// Check ParCmd.ProcessingMode defined ? 
IF (( ProcessingMode < ProcessingModeEnum.BUFFERED         ) AND
    ( ProcessingMode > ProcessingModeEnum.TRIGGER_MULTIPLE ))
THEN
  // Parameter not valid
  CheckParameterValid := FALSE;
  // Set error
  SetError( ErrorID := RobotLibraryErrorIdEnum.ERR_PROCESSINGMODE_NOT_DEFINED, Overwrite := TRUE );
  // Create log entry
  CreateLogMessagePara1 ( Timestamp   := AxesGroup.State.SystemTime,
                          MessageType := MessageType.CMD,
                          Severity    := Severity.ERROR,
                          MessageCode := ErrorID,
                          MessageText := 'Invalid Parameter ParCmd.ProcessingMode = {1}',
                          Para1       := PROCESSING_MODE_TO_STRING(ProcessingMode));
  RETURN;                          
END_IF


// Check ProcessingMode valid ? 
IF (( ProcessingMode <> ProcessingModeEnum.BUFFERED           ) AND
    ( ProcessingMode <> ProcessingModeEnum.ABORTING           ) AND  
    ( ProcessingMode <> ProcessingModeEnum.PARALLEL           ) AND
    ( ProcessingMode <> ProcessingModeEnum.CONTINUOUS         ) AND
    ( ProcessingMode <> ProcessingModeEnum.DEACTIVATE         ) AND
    ( ProcessingMode <> ProcessingModeEnum.TRIGGER_ONCE       ) AND
    ( ProcessingMode <> ProcessingModeEnum.TRIGGER_CONTINUOUS ) AND
    ( ProcessingMode <> ProcessingModeEnum.TRIGGER_MULTIPLE   )) 
THEN
  // Parameter not valid
  CheckParameterValid := FALSE;
  // Set error
  SetError( ErrorID := RobotLibraryErrorIdEnum.ERR_PROCESSINGMODE_NOT_ALLOWED, Overwrite := TRUE );
  // Create log entry
  CreateLogMessagePara1 ( Timestamp   := AxesGroup.State.SystemTime,
                          MessageType := MessageType.CMD,
                          Severity    := Severity.ERROR,
                          MessageCode := ErrorID,
                          MessageText := 'Invalid Parameter ProcessingMode = {1}',
                          Para1       := PROCESSING_MODE_TO_STRING(ProcessingMode));
  RETURN;                          
END_IF

// Check SequenceFlag valid ? 
IF (( SequenceFlag <> SequenceFlagEnum.NO_SEQUENCE        ) AND    
    ( SequenceFlag <> SequenceFlagEnum.PRIMARY_SEQUENCE   ) AND
    ( SequenceFlag <> SequenceFlagEnum.SECONDARY_SEQUENCE ))
THEN
  // Parameter not valid
  CheckParameterValid := FALSE;
  // Set error
  SetError( ErrorID := RobotLibraryErrorIdEnum.ERR_SEQFLAG_NOT_ALLOWED, Overwrite := TRUE );
  // Create log entry
  CreateLogMessagePara1 ( Timestamp   := AxesGroup.State.SystemTime,
                          MessageType := MessageType.CMD,
                          Severity    := Severity.ERROR,
                          MessageCode := ErrorID,
                          MessageText := 'Invalid Parameter SequenceFlag = {1}',
                          Para1       := SEQUENCE_FLAG_TO_STRING(SequenceFlag));
  RETURN;                          
END_IF


// Check ParCmd.JobID valid ? 
IF (( ParCmd.JobID <     0 ) OR  
    ( ParCmd.JobID > 65535 ))
THEN
  // Parameter not valid
  CheckParameterValid := FALSE;
  // Set error
  SetError( ErrorID := RobotLibraryErrorIdEnum.ERR_LISTENERID_MUST_BE_POSITIVE, Overwrite := TRUE );
  // Create log entry
  CreateLogMessagePara1 ( Timestamp   := AxesGroup.State.SystemTime,
                          MessageType := MessageType.CMD,
                          Severity    := Severity.ERROR,
                          MessageCode := ErrorID,
                          MessageText := 'Invalid Parameter ParCmd.JobID = {1}',
                          Para1       := UINT_TO_STRING(ParCmd.JobID));
  RETURN;                          
END_IF


// Check ParCmd.ListenerID valid ? 
IF (( ParCmd.ListenerID <   0 ) OR  
    ( ParCmd.ListenerID > 127 ))
THEN
  // Parameter not valid
  CheckParameterValid := FALSE;
  // Set error
  SetError( ErrorID := RobotLibraryErrorIdEnum.ERR_LISTENERID_MUST_BE_POSITIVE, Overwrite := TRUE );
  // Create log entry
  CreateLogMessagePara1 ( Timestamp   := AxesGroup.State.SystemTime,
                          MessageType := MessageType.CMD,
                          Severity    := Severity.ERROR,
                          MessageCode := ErrorID,
                          MessageText := 'Invalid Parameter ParCmd.ListenerID = {1}',
                          Para1       := SINT_TO_STRING(ParCmd.ListenerID));
  RETURN;                          
END_IF



FOR _idx := 0 TO RobotLibraryParameter.SUB_PROGRAM_DATA_MAX
DO
  // Check ParCmd.Data valid ? 
  IF (( ParCmd.Data[_idx] <   0 ) OR  
      ( ParCmd.Data[_idx] > 255 ))
  THEN
    // Parameter not valid
    CheckParameterValid := FALSE;
    // Set error
    SetError( ErrorID := RobotLibraryErrorIdEnum.ERR_LISTENERID_MUST_BE_POSITIVE, Overwrite := TRUE );
    // Create log entry
    CreateLogMessagePara2 ( Timestamp   := AxesGroup.State.SystemTime,
                            MessageType := MessageType.CMD,
                            Severity    := Severity.ERROR,
                            MessageCode := ErrorID,
                            MessageText := 'Invalid Parameter ParCmd.Data[{2}] = {1}',
                            Para1       := BYTE_TO_STRING(ParCmd.Data[_idx]),
                            Para2       := DINT_TO_STRING(_idx));
    EXIT;                            
    RETURN;                          
  END_IF
END_FOR
                
END_METHOD

METHOD INTERNAL CreateCommandPayload : RobotLibraryCommandDataFB
VAR_IN_OUT
  /// Robot assignment of function
  AxesGroup : AxesGroup; 
END_VAR
VAR
  /// internal index for loops
 _idx          : DINT;
  /// Parameter count
 _parameterCnt : DINT;
END_VAR// Table 6-687: Sent CMD payload (PLC to RC) of "CallSubprogram"
// --------------------------
// Header
// --------------------------
// Byte 00 : UINT  - Type HB     
// Byte 01 :       - Type LB    
// Byte 02 : USINT - Reserve | ExecutionMode
// Byte 03 : USINT - ParSeq  | Priority
// --------------------------
// Datablock
// --------------------------
// Byte 00 : UINT  Type;
// Byte 01 :       Type;
// Byte 02 : USINT Reserved ExecutionMode;
// Byte 03 : USINT ParSeq Priority;
// Byte 04 : SINT  EmitterID[0];
// Byte 05 : SINT  EmitterID[1];
// Byte 06 : SINT  EmitterID[2];
// Byte 07 : SINT  EmitterID[3];
// Byte 08 : SINT  ListenerID;
// Byte 09 : BYTE  Reserved;
// Byte 10 : UINT  JobID;
// Byte 11 :       JobID;
// Byte 12 : BYTE  Data[0];
// Byte 13 : BYTE  Data[1];
// Byte 14 : BYTE  Data[2];
// Byte 15 : BYTE  Data[3];
// Byte 16 : BYTE  Data[4];
// Byte 17 : BYTE  Data[5];
// Byte 18 : BYTE  Data[6];
// Byte 19 : BYTE  Data[7];
// Byte 20 : BYTE  Data[8];
// Byte 21 : BYTE  Data[9];
// Byte 22 : BYTE  Data[10];
// Byte 23 : BYTE  Data[11];
// Byte 24 : BYTE  Data[12];
// Byte 25 : BYTE  Data[13];
// Byte 26 : BYTE  Data[14];
// Byte 27 : BYTE  Data[15];
// Byte 28 : BYTE  Data[16];
// Byte 29 : BYTE  Data[17];
// Byte 30 : BYTE  Data[18];
// Byte 31 : BYTE  Data[19];
// Byte 32 : BYTE  Data[20];
// Byte 33 : BYTE  Data[21];
// Byte 34 : BYTE  Data[22];
// Byte 35 : BYTE  Data[23];
// Byte 36 : BYTE  Data[24];
// Byte 37 : BYTE  Data[25];
// Byte 38 : BYTE  Data[26];
// Byte 39 : BYTE  Data[27];
// Byte 40 : BYTE  Data[28];
// Byte 41 : BYTE  Data[29];
// Byte 42 : BYTE  Data[30];
// Byte 43 : BYTE  Data[31];
// Byte 44 : BYTE  Data[32];
// Byte 45 : BYTE  Data[33];
// Byte 46 : BYTE  Data[34];
// Byte 47 : BYTE  Data[35];
// Byte 48 : BYTE  Data[36];
// Byte 49 : BYTE  Data[37];
// Byte 50 : BYTE  Data[38];
// Byte 51 : BYTE  Data[39];
// Byte 52 : BYTE  Data[40];
// Byte 53 : BYTE  Data[41];
// Byte 54 : BYTE  Data[42];
// Byte 55 : BYTE  Data[43];
// Byte 56 : BYTE  Data[44];
// Byte 57 : BYTE  Data[45];
// Byte 58 : BYTE  Data[46];
// Byte 59 : BYTE  Data[47];
// Byte 60 : BYTE  Data[48];
// Byte 61 : BYTE  Data[49];
// Byte 62 : BYTE  Data[50];
// Byte 63 : BYTE  Data[51];
// Byte 64 : BYTE  Data[52];
// Byte 65 : BYTE  Data[53];
// Byte 66 : BYTE  Data[54];
// Byte 67 : BYTE  Data[55];
// Byte 68 : BYTE  Data[56];
// Byte 69 : BYTE  Data[57];
// Byte 70 : BYTE  Data[58];
// Byte 71 : BYTE  Data[59];
// Byte 72 : BYTE  Data[60];
// Byte 73 : BYTE  Data[61];
// Byte 74 : BYTE  Data[62];
// Byte 75 : BYTE  Data[63];
// Byte 76 : BYTE  Data[64];
// Byte 77 : BYTE  Data[65];
// Byte 78 : BYTE  Data[66];
// Byte 79 : BYTE  Data[67];
// Byte 80 : BYTE  Data[68];
// Byte 81 : BYTE  Data[69];
// Byte 82 : BYTE  Data[70];
// Byte 83 : BYTE  Data[71];
// Byte 84 : BYTE  Data[72];
// Byte 85 : BYTE  Data[73];
// Byte 86 : BYTE  Data[74];
// Byte 87 : BYTE  Data[75];
// Byte 88 : BYTE  Data[76];
// Byte 89 : BYTE  Data[77];
// Byte 90 : BYTE  Data[78];
// Byte 91 : BYTE  Data[79];
// Byte 92 : BYTE  Data[80];
// Byte 93 : BYTE  Data[81];
// Byte 94 : BYTE  Data[82];
// Byte 95 : BYTE  Data[83];
// Byte 96 : BYTE  Data[84];
// Byte 97 : BYTE  Data[85];
// Byte 98 : BYTE  Data[86];
// Byte 99 : BYTE  Data[87];
// Byte 100: BYTE  Data[88];
// Byte 101: BYTE  Data[89];
// Byte 102: BYTE  Data[90];
// Byte 103: BYTE  Data[91];
// Byte 104: BYTE  Data[92];
// Byte 105: BYTE  Data[93];
// Byte 106: BYTE  Data[94];
// Byte 107: BYTE  Data[95];
// Byte 108: BYTE  Data[96];
// Byte 109: BYTE  Data[97];
// Byte 110: BYTE  Data[98];
// Byte 111: BYTE  Data[99];
// Byte 112: BYTE  Data[100];
// Byte 113: BYTE  Data[101];
// Byte 114: BYTE  Data[102];
// Byte 115: BYTE  Data[103];
// Byte 116: BYTE  Data[104];
// Byte 117: BYTE  Data[105];
// Byte 118: BYTE  Data[106];
// Byte 119: BYTE  Data[107];
// Byte 120: BYTE  Data[108];
// Byte 121: BYTE  Data[109];
// Byte 122: BYTE  Data[110];
// Byte 123: BYTE  Data[111];
// Byte 124: BYTE  Data[112];
// Byte 125: BYTE  Data[113];
// Byte 126: BYTE  Data[114];
// Byte 127: BYTE  Data[115];
// Byte 128: BYTE  Data[116];
// Byte 129: BYTE  Data[117];
// Byte 130: BYTE  Data[118];
// Byte 131: BYTE  Data[119];
// Byte 132: BYTE  Data[120];
// Byte 133: BYTE  Data[121];
// Byte 134: BYTE  Data[122];
// Byte 135: BYTE  Data[123];
// Byte 136: BYTE  Data[124];
// Byte 137: BYTE  Data[125];
// Byte 138: BYTE  Data[126];
// Byte 139: BYTE  Data[127];
// Byte 140: BYTE  Data[128];
// Byte 141: BYTE  Data[129];
// Byte 142: BYTE  Data[130];
// Byte 143: BYTE  Data[131];
// Byte 144: BYTE  Data[132];
// Byte 145: BYTE  Data[133];
// Byte 146: BYTE  Data[134];
// Byte 147: BYTE  Data[135];
// Byte 148: BYTE  Data[136];
// Byte 149: BYTE  Data[137];
// Byte 150: BYTE  Data[138];
// Byte 151: BYTE  Data[139];
// Byte 152: BYTE  Data[140];
// Byte 153: BYTE  Data[141];
// Byte 154: BYTE  Data[142];
// Byte 155: BYTE  Data[143];
// Byte 156: BYTE  Data[144];
// Byte 157: BYTE  Data[145];
// Byte 158: BYTE  Data[146];
// Byte 159: BYTE  Data[147];
// Byte 160: BYTE  Data[148];
// Byte 161: BYTE  Data[149];
// Byte 162: BYTE  Data[150];
// Byte 163: BYTE  Data[151];
// Byte 164: BYTE  Data[152];
// Byte 165: BYTE  Data[153];
// Byte 166: BYTE  Data[154];
// Byte 167: BYTE  Data[155];
// Byte 168: BYTE  Data[156];
// Byte 169: BYTE  Data[157];
// Byte 170: BYTE  Data[158];
// Byte 171: BYTE  Data[159];
// Byte 172: BYTE  Data[160];
// Byte 173: BYTE  Data[161];
// Byte 174: BYTE  Data[162];
// Byte 175: BYTE  Data[163];
// Byte 176: BYTE  Data[164];
// Byte 177: BYTE  Data[165];
// Byte 178: BYTE  Data[166];
// Byte 179: BYTE  Data[167];
// Byte 180: BYTE  Data[168];
// Byte 181: BYTE  Data[169];
// Byte 182: BYTE  Data[170];
// Byte 183: BYTE  Data[171];
// Byte 184: BYTE  Data[172];
// Byte 185: BYTE  Data[173];
// Byte 186: BYTE  Data[174];
// Byte 187: BYTE  Data[175];
// Byte 188: BYTE  Data[176];
// Byte 189: BYTE  Data[177];
// Byte 190: BYTE  Data[178];
// Byte 191: BYTE  Data[179];
// Byte 192: BYTE  Data[180];
// Byte 193: BYTE  Data[181];
// Byte 194: BYTE  Data[182];
// Byte 195: BYTE  Data[183];
// Byte 196: BYTE  Data[184];
// Byte 197: BYTE  Data[185];
// Byte 198: BYTE  Data[186];
// Byte 199: BYTE  Data[187];
// Byte 200: BYTE  Data[188];
// Byte 201: BYTE  Data[189];
                  // set command parameter 
_command.CmdTyp       :=  CmdType.CallSubprogram;
_command.ExecMode     :=  ExecMode;
_command.ParSeq       := _command.ParSeq;
_command.Priority     :=  Priority;
_command.EmitterID[0] :=  0;
_command.EmitterID[1] :=  0;
_command.EmitterID[2] :=  0;
_command.EmitterID[3] :=  0;
_command.Reserve      :=  0;
_command.ListenerID   := _parCmd.ListenerID;
_command.Reserve      := 0;
_command.JobID        := _parCmd.JobID;
_command.Data         := _parCmd.Data;


// copy command data to header
_cmdHeader := _command;
// call base implementation to copy header to payload buffer
CreateCommandPayload := SUPER^.CreateCommandPayload(AxesGroup := AxesGroup);


FOR _idx := 0 TO 3
DO
  // Check parameter must be added ? 
  IF ( CheckAddParameter(CreateCommandPayload.PayloadPtr))
  THEN
    // add command.EmitterID
    CreateCommandPayload.AddSint(_command.EmitterID[_idx]);
    // inc parameter counter
   _parameterCnt := _parameterCnt + 1;  
  END_IF
END_FOR


// Check parameter must be added ? 
IF ( CheckAddParameter(CreateCommandPayload.PayloadPtr))
THEN
  // add command.ListenerID
  CreateCommandPayload.AddSint(_command.ListenerID);
  // inc parameter counter
 _parameterCnt := _parameterCnt + 1;  
END_IF


// Check parameter must be added ? 
IF ( CheckAddParameter(CreateCommandPayload.PayloadPtr))
THEN
  // add command.Reserve
  CreateCommandPayload.AddByte(_command.Reserve);
  // inc parameter counter
 _parameterCnt := _parameterCnt + 1;  
END_IF


// Check parameter must be added ? 
IF ( CheckAddParameter(CreateCommandPayload.PayloadPtr))
THEN
  // add command.JobID
  CreateCommandPayload.AddUint(_command.JobID);
  // inc parameter counter
 _parameterCnt := _parameterCnt + 1;  
END_IF
  
  
FOR _idx := 0 TO RobotLibraryParameter.SUB_PROGRAM_DATA_MAX
DO
  // Check parameter must be added ? 
  IF ( CheckAddParameter(CreateCommandPayload.PayloadPtr))
  THEN
    // add command.Data[_idx]
    CreateCommandPayload.AddByte(_command.Data[_idx]);
    // inc parameter counter
   _parameterCnt := _parameterCnt + 1;  
  END_IF
END_FOR


// Create logging
CreateCommandPayloadLog(AxesGroup := AxesGroup, ParameterCnt := _parameterCnt);
                
END_METHOD

METHOD INTERNAL CreateCommandPayloadLog
VAR_IN_OUT
  /// Robot assignment of function
  AxesGroup : AxesGroup; 
END_VAR
VAR_INPUT
  /// Parameter count
  ParameterCnt : DINT;
END_VAR
VAR
  /// internal index for loops
 _idx : DINT;
END_VAR
                  // Create log entry for Parameter start
CreateLogMessagePara1 ( Timestamp   := AxesGroup.State.SystemTime,
                        MessageType := MessageType.CMD,
                        Severity    := Severity.DEBUG,
                        MessageCode := 0,
                        MessageText := 'Create command payload with {1} parameter(s) :',
                        Para1       := DINT_TO_STRING(ParameterCnt));
  
// Create log entry for EmitterID[x]
FOR _idx := 0 TO 3
DO
  // Return if no parameter is remaining...
  IF ( ParameterCnt = 0 ) THEN RETURN; END_IF
  // dec remaining parameter(s)                        
  ParameterCnt := ParameterCnt - 1;
  // Create log entry for Command.EmitterID
  CreateLogMessagePara2 ( Timestamp   := AxesGroup.State.SystemTime,
                          MessageType := MessageType.CMD,
                          Severity    := Severity.DEBUG,
                          MessageCode := 0,
                          MessageText := 'Command.EmitterID[{2}] = {1}',
                          Para1       :=  SINT_TO_STRING(_command.EmitterID[_idx]),
                          Para2       :=  DINT_TO_STRING(_idx));
END_FOR


// Return if no parameter is remaining...
IF ( ParameterCnt = 0 ) THEN RETURN; END_IF
// dec remaining parameter(s)                        
ParameterCnt := ParameterCnt - 1;
// Create log entry for ListenerID
CreateLogMessagePara1 ( Timestamp   := AxesGroup.State.SystemTime,
                        MessageType := MessageType.CMD,
                        Severity    := Severity.DEBUG,
                        MessageCode := 0,
                        MessageText := 'Command.ListenerID = {1}',
                        Para1       :=  SINT_TO_STRING(_command.ListenerID));


// Return if no parameter is remaining...
IF ( ParameterCnt = 0 ) THEN RETURN; END_IF
// dec remaining parameter(s)                        
ParameterCnt := ParameterCnt - 1;
// Create log entry for Reserve
CreateLogMessagePara1 ( Timestamp   := AxesGroup.State.SystemTime,
                        MessageType := MessageType.CMD,
                        Severity    := Severity.DEBUG,
                        MessageCode := 0,
                        MessageText := 'Command.Reserve = {1}',
                        Para1       :=  BYTE_TO_STRING(_command.Reserve));


// Return if no parameter is remaining...
IF ( ParameterCnt = 0 ) THEN RETURN; END_IF
// dec remaining parameter(s)                        
ParameterCnt := ParameterCnt - 1;
// Create log entry for JobID
CreateLogMessagePara1 ( Timestamp   := AxesGroup.State.SystemTime,
                        MessageType := MessageType.CMD,
                        Severity    := Severity.DEBUG,
                        MessageCode := 0,
                        MessageText := 'Command.JobID = {1}',
                        Para1       :=  UINT_TO_STRING(_command.JobID));


FOR _idx := 0 TO RobotLibraryParameter.SUB_PROGRAM_DATA_MAX
DO
  // Return if no parameter is remaining...
  IF ( ParameterCnt = 0 ) THEN RETURN; END_IF
  // dec remaining parameter(s)                        
  ParameterCnt := ParameterCnt - 1;
  // Create log entry for Data
  CreateLogMessagePara1 ( Timestamp   := AxesGroup.State.SystemTime,
                          MessageType := MessageType.CMD,
                          Severity    := Severity.DEBUG,
                          MessageCode := 0,
                          MessageText := StrReplace('Command.Data[{0}] = {1}', '{0}', DINT_TO_STRING(_idx)), 
                          Para1       :=  UINT_TO_STRING(_command.Data[_idx]));
END_FOR
                
END_METHOD

METHOD FB_init : BOOL
VAR_INPUT
  /// if TRUE, the retain variables are initialized (warm start / cold start)
  bInitRetains : BOOL; 
  /// if TRUE, the instance afterwards gets moved into the copy code (online change)
  bInCopyCode  : BOOL;  
END_VAR
                  MyType := 'MC_CallSubprogramFB';

ExecMode       := ExecutionMode.PARALLEL;
Priority       := PriorityLevel.NORMAL;
ProcessingMode := ProcessingModeEnum.PARALLEL;
SequenceFlag   := SequenceFlagEnum.NO_SEQUENCE;  

                
END_METHOD

METHOD PROTECTED OnApplyOutCmd
VAR_INPUT
  /// Command message state
  State : CmdMessageState;
END_VAR
                  IF ( State = CmdMessageState.EMPTY ) 
THEN
  // Reset command outputs
  SysDepMemSet(pDest := ADR(OutCmd), Value := 0, DataLen := SIZEOF(OutCmd));         
END_IF

IF ( State = CmdMessageState.DONE )
THEN
  // Update results
  OutCmd.InstanceID        := 0; {warning 'ToDo'}
  OutCmd.OriginID          := _response.OriginID;
  OutCmd.InvocationCounter := _response.InvocationCounter;
  OutCmd.ReturnData        := _response.ReturnData;
END_IF
                
END_METHOD

METHOD PROTECTED OnExecRun : DINT
VAR_IN_OUT
  /// Robot assignment of function
  AxesGroup : AxesGroup; 
END_VAR
                  // call base implementation
SUPER^.OnExecRun(AxesGroup := AxesGroup);

CASE _stepCmd OF
  
  00:  IF ( _execute_R.Q ) AND ( NOT Error)  
       THEN
         // Check function is supported and parameter are valid ?
         IF (( CheckFunctionSupported( AxesGroup := AxesGroup )) AND
             ( CheckParameterValid   ( AxesGroup := AxesGroup )))      
         THEN
           // set busy flag
           Busy := TRUE;
           // Reset command outputs
           SysDepMemSet(pDest := ADR(OutCmd), Value := 0, DataLen := SIZEOF(OutCmd));         
           // apply command parameter
          _parCmd := ParCmd;
           // init parameter sequence
          _command.ParSeq := 1;
           // create command data
           CommandData := CreateCommandPayload(AxesGroup := AxesGroup);
           // Add command to active command register
          _uniqueID := AxesGroup.Acyclic.ActiveCommandRegister.AddCmd( pCommandFB := ADR(THIS^ ));     
           // set timeout
           SetTimeout(PT := _timeoutCmd, rTimer := _timerCmd);
           // inc step counter
          _stepCmd := _stepCmd + 1; 
          END_IF
       END_IF
     

  01:  // Wait for responce received
       IF ( _responseReceived )
       THEN
         // reset response received flag
        _responseReceived := FALSE;
         // update state flags
         OnUpdateStateFlags(_response.State);
         // update state flags
         OnApplyOutCmd(_response.State);
         
         // Done, Aborted or Error ?
         IF (_response.State >= CmdMessageState.DONE )
         THEN
           // set timeout
           SetTimeout(PT := _timeoutCmd, rTimer := _timerCmd);
           // inc step counter
          _stepCmd := _stepCmd + 1; 
         END_IF
       END_IF


  02: IF ( NOT Execute)
      THEN
        Reset();
      END_IF     
ELSE
  // invalid step
  SetError( ErrorID := RobotLibraryErrorIdEnum.ERR_INVALID_STEP, Overwrite := TRUE );
END_CASE



// Reset FB
IF ( NOT Execute )
THEN
  Reset();  
END_IF
                
END_METHOD

METHOD PROTECTED OnUpdateStateFlags
VAR_INPUT
  /// Command message state
  State : CmdMessageState;
END_VAR
                  // Reset State flags
CommandAborted     := FALSE;
CommandInterrupted := FALSE;
Done               := FALSE;

// Update in prograss value
InProgress := _response.InProgress;

CASE State OF

  // No operation or process is active
  CmdMessageState.EMPTY               :;
  // Created but not yet started
  CmdMessageState.CREATED             :;
  // Buffered and awaiting execution
  CmdMessageState.BUFFERED            : CommandBuffered    := TRUE;
  // Buffered in planner for future execution
  CmdMessageState.BUFFERED_IN_PLANNER : CommandBuffered    := TRUE;
  // Currently active and in progress
  CmdMessageState.ACTIVE              :;
  // Interrupted and awaiting continuation
  CmdMessageState.INTERRUPTED         : CommandInterrupted := TRUE;
  // Requested for abort
  CmdMessageState.ABORT_REQUEST       :;
  // Successfully completed
  CmdMessageState.DONE                : Done               := TRUE;
                                        Busy               := FALSE;
  // Aborted before completion
  CmdMessageState.ABORTED             : CommandAborted     := TRUE;
                                        Busy               := FALSE;
  // Encountered an error during execution
  CmdMessageState.ERROR               : Error              := TRUE;
                                        Busy               := FALSE;
END_CASE
                
END_METHOD

METHOD INTERNAL ParseResponsePayload : DINT
VAR_INPUT
  /// Response data
  ResponseData : RobotLibraryResponseDataFB;
  /// Timestamp
  Timestamp    : SystemTime;  
END_VAR
VAR
  /// internal index for loops
 _idx          : DINT;
  /// Parameter count
 _parameterCnt : DINT;
END_VAR
// Table 6-688: Received CMD payload (RC to PLC) of "CallSubprogram"
// --------------------------
// Header
// --------------------------
// Byte 00 : USINT   - ParSeq | State     
// Byte 01 : SINT    - AlarmMessageSeverity    
// Byte 02 : UINT    - AlarmMessageCode HB
// Byte 03 :         - AlarmMessageCode LB
// --------------------------
// Datablock
// --------------------------
// Byte 04 : USINT InvocationCounter;
// Byte 05 : SINT  Reserved;
// Byte 06 : INT   OriginID;
// Byte 07 :       OriginID;
// Byte 08 : UINT  Progress;
// Byte 09 :       Progress;
// Byte 10 : BOOL  InProgress;
// Byte 11 : BYTE  ReturnData[0];
// Byte 12 : BYTE  ReturnData[1];
// Byte 13 : BYTE  ReturnData[2];
// Byte 14 : BYTE  ReturnData[3];
// Byte 15 : BYTE  ReturnData[4];
// Byte 16 : BYTE  ReturnData[5];
// Byte 17 : BYTE  ReturnData[6];
// Byte 18 : BYTE  ReturnData[7];
// Byte 19 : BYTE  ReturnData[8];
// Byte 20 : BYTE  ReturnData[9];
// Byte 21 : BYTE  ReturnData[10];
// Byte 22 : BYTE  ReturnData[11];
// Byte 23 : BYTE  ReturnData[12];
// Byte 24 : BYTE  ReturnData[13];
// Byte 25 : BYTE  ReturnData[14];
// Byte 26 : BYTE  ReturnData[15];
// Byte 27 : BYTE  ReturnData[16];
// Byte 28 : BYTE  ReturnData[17];
// Byte 29 : BYTE  ReturnData[18];
// Byte 30 : BYTE  ReturnData[19];
// Byte 31 : BYTE  ReturnData[20];
// Byte 32 : BYTE  ReturnData[21];
// Byte 33 : BYTE  ReturnData[22];
// Byte 34 : BYTE  ReturnData[23];
// Byte 35 : BYTE  ReturnData[24];
// Byte 36 : BYTE  ReturnData[25];
// Byte 37 : BYTE  ReturnData[26];
// Byte 38 : BYTE  ReturnData[27];
// Byte 39 : BYTE  ReturnData[28];
// Byte 40 : BYTE  ReturnData[29];
// Byte 41 : BYTE  ReturnData[30];
// Byte 42 : BYTE  ReturnData[31];
// Byte 43 : BYTE  ReturnData[32];
// Byte 44 : BYTE  ReturnData[33];
// Byte 45 : BYTE  ReturnData[34];
// Byte 46 : BYTE  ReturnData[35];
// Byte 47 : BYTE  ReturnData[36];
// Byte 48 : BYTE  ReturnData[37];
// Byte 49 : BYTE  ReturnData[38];
// Byte 50 : BYTE  ReturnData[39];
// Byte 51 : BYTE  ReturnData[40];
// Byte 52 : BYTE  ReturnData[41];
// Byte 53 : BYTE  ReturnData[42];
// Byte 54 : BYTE  ReturnData[43];
// Byte 55 : BYTE  ReturnData[44];
// Byte 56 : BYTE  ReturnData[45];
// Byte 57 : BYTE  ReturnData[46];
// Byte 58 : BYTE  ReturnData[47];
// Byte 59 : BYTE  ReturnData[48];
// Byte 60 : BYTE  ReturnData[49];
// Byte 61 : BYTE  ReturnData[50];
// Byte 62 : BYTE  ReturnData[51];
// Byte 63 : BYTE  ReturnData[52];
// Byte 64 : BYTE  ReturnData[53];
// Byte 65 : BYTE  ReturnData[54];
// Byte 66 : BYTE  ReturnData[55];
// Byte 67 : BYTE  ReturnData[56];
// Byte 68 : BYTE  ReturnData[57];
// Byte 69 : BYTE  ReturnData[58];
// Byte 70 : BYTE  ReturnData[59];
// Byte 71 : BYTE  ReturnData[60];
// Byte 72 : BYTE  ReturnData[61];
// Byte 73 : BYTE  ReturnData[62];
// Byte 74 : BYTE  ReturnData[63];
// Byte 75 : BYTE  ReturnData[64];
// Byte 76 : BYTE  ReturnData[65];
// Byte 77 : BYTE  ReturnData[66];
// Byte 78 : BYTE  ReturnData[67];
// Byte 79 : BYTE  ReturnData[68];
// Byte 80 : BYTE  ReturnData[69];
// Byte 81 : BYTE  ReturnData[70];
// Byte 82 : BYTE  ReturnData[71];
// Byte 83 : BYTE  ReturnData[72];
// Byte 84 : BYTE  ReturnData[73];
// Byte 85 : BYTE  ReturnData[74];
// Byte 86 : BYTE  ReturnData[75];
// Byte 87 : BYTE  ReturnData[76];
// Byte 88 : BYTE  ReturnData[77];
// Byte 89 : BYTE  ReturnData[78];
// Byte 90 : BYTE  ReturnData[79];
// Byte 91 : BYTE  ReturnData[80];
// Byte 92 : BYTE  ReturnData[81];
// Byte 93 : BYTE  ReturnData[82];
// Byte 94 : BYTE  ReturnData[83];
// Byte 95 : BYTE  ReturnData[84];
// Byte 96 : BYTE  ReturnData[85];
// Byte 97 : BYTE  ReturnData[86];
// Byte 98 : BYTE  ReturnData[87];
// Byte 99 : BYTE  ReturnData[88];
// Byte 100: BYTE  ReturnData[89];
// Byte 101: BYTE  ReturnData[90];
// Byte 102: BYTE  ReturnData[91];
// Byte 103: BYTE  ReturnData[92];
// Byte 104: BYTE  ReturnData[93];
// Byte 105: BYTE  ReturnData[94];
// Byte 106: BYTE  ReturnData[95];
// Byte 107: BYTE  ReturnData[96];
// Byte 108: BYTE  ReturnData[97];
// Byte 109: BYTE  ReturnData[98];
// Byte 110: BYTE  ReturnData[99];
// Byte 111: BYTE  ReturnData[100];
// Byte 112: BYTE  ReturnData[101];
// Byte 113: BYTE  ReturnData[102];
// Byte 114: BYTE  ReturnData[103];
// Byte 115: BYTE  ReturnData[104];
// Byte 116: BYTE  ReturnData[105];
// Byte 117: BYTE  ReturnData[106];
// Byte 118: BYTE  ReturnData[107];
// Byte 119: BYTE  ReturnData[108];
// Byte 120: BYTE  ReturnData[109];
// Byte 121: BYTE  ReturnData[110];
// Byte 122: BYTE  ReturnData[111];
// Byte 123: BYTE  ReturnData[112];
// Byte 124: BYTE  ReturnData[113];
// Byte 125: BYTE  ReturnData[114];
// Byte 126: BYTE  ReturnData[115];
// Byte 127: BYTE  ReturnData[116];
// Byte 128: BYTE  ReturnData[117];
// Byte 129: BYTE  ReturnData[118];
// Byte 130: BYTE  ReturnData[119];
// Byte 131: BYTE  ReturnData[120];
// Byte 132: BYTE  ReturnData[121];
// Byte 133: BYTE  ReturnData[122];
// Byte 134: BYTE  ReturnData[123];
// Byte 135: BYTE  ReturnData[124];
// Byte 136: BYTE  ReturnData[125];
// Byte 137: BYTE  ReturnData[126];
// Byte 138: BYTE  ReturnData[127];
// Byte 139: BYTE  ReturnData[128];
// Byte 140: BYTE  ReturnData[129];
// Byte 141: BYTE  ReturnData[130];
// Byte 142: BYTE  ReturnData[131];
// Byte 143: BYTE  ReturnData[132];
// Byte 144: BYTE  ReturnData[133];
// Byte 145: BYTE  ReturnData[134];
// Byte 146: BYTE  ReturnData[135];
// Byte 147: BYTE  ReturnData[136];
// Byte 148: BYTE  ReturnData[137];
// Byte 149: BYTE  ReturnData[138];
// Byte 150: BYTE  ReturnData[139];
// Byte 151: BYTE  ReturnData[140];
// Byte 152: BYTE  ReturnData[141];
// Byte 153: BYTE  ReturnData[142];
// Byte 154: BYTE  ReturnData[143];
// Byte 155: BYTE  ReturnData[144];
// Byte 156: BYTE  ReturnData[145];
// Byte 157: BYTE  ReturnData[146];
// Byte 158: BYTE  ReturnData[147];
// Byte 159: BYTE  ReturnData[148];
// Byte 160: BYTE  ReturnData[149];
// Byte 161: BYTE  ReturnData[150];
// Byte 162: BYTE  ReturnData[151];
// Byte 163: BYTE  ReturnData[152];
// Byte 164: BYTE  ReturnData[153];
// Byte 165: BYTE  ReturnData[154];
// Byte 166: BYTE  ReturnData[155];
// Byte 167: BYTE  ReturnData[156];
// Byte 168: BYTE  ReturnData[157];
// Byte 169: BYTE  ReturnData[158];
// Byte 170: BYTE  ReturnData[159];
// Byte 171: BYTE  ReturnData[160];
// Byte 172: BYTE  ReturnData[161];
// Byte 173: BYTE  ReturnData[162];
// Byte 174: BYTE  ReturnData[163];
// Byte 175: BYTE  ReturnData[164];
// Byte 176: BYTE  ReturnData[165];
// Byte 177: BYTE  ReturnData[166];
// Byte 178: BYTE  ReturnData[167];
// Byte 179: BYTE  ReturnData[168];
// Byte 180: BYTE  ReturnData[169];
// Byte 181: BYTE  ReturnData[170];
// Byte 182: BYTE  ReturnData[171];
// Byte 183: BYTE  ReturnData[172];
// Byte 184: BYTE  ReturnData[173];
// Byte 185: BYTE  ReturnData[174];
// Byte 186: BYTE  ReturnData[175];
// Byte 187: BYTE  ReturnData[176];
// Byte 188: BYTE  ReturnData[177];
// Byte 189: BYTE  ReturnData[178];
// Byte 190: BYTE  ReturnData[179];
// Byte 191: BYTE  ReturnData[180];
// Byte 192: BYTE  ReturnData[181];
// Byte 193: BYTE  ReturnData[182];
// Byte 194: BYTE  ReturnData[183];
// Byte 195: BYTE  ReturnData[184];
// Byte 196: BYTE  ReturnData[185];
// Byte 197: BYTE  ReturnData[186];
// Byte 198: BYTE  ReturnData[187];
// Byte 199: BYTE  ReturnData[188];
// Byte 200: BYTE  ReturnData[189];
                  // call base implementation to parse the header from payload buffer
ResponseData.PayloadPtr := SUPER^.ParseResponsePayload(ResponseData := ResponseData, Timestamp := Timestamp);

// copy parsed header to response
_response.ParSeq               := _rspHeader.ParSeq;
_response.State                := _rspHeader.State;
_response.AlarmMessageSeverity := _rspHeader.AlarmMessageSeverity;
_response.AlarmMessageCode     := _rspHeader.AlarmMessageCode;


// Check payload remaining ? 
IF ( ResponseData.IsPayloadRemaining)
THEN
  // Get Response.InvocationCounter
 _response.InvocationCounter := ResponseData.GetUsint();
  // inc parameter counter
 _parameterCnt := _parameterCnt + 1;
END_IF


// Check payload remaining ? 
IF ( ResponseData.IsPayloadRemaining)
THEN
  // Get Response.Reserve
 _response.Reserve := ResponseData.GetSint();
  // inc parameter counter
 _parameterCnt := _parameterCnt + 1;
END_IF


// Check payload remaining ? 
IF ( ResponseData.IsPayloadRemaining)
THEN
  // Get Response.OriginID
 _response.OriginID := ResponseData.GetInt();
  // inc parameter counter
 _parameterCnt := _parameterCnt + 1;
END_IF


// Check payload remaining ? 
IF ( ResponseData.IsPayloadRemaining)
THEN
  // Get Response.Progress
 _response.Progress := ResponseData.GetUint();
  // inc parameter counter
 _parameterCnt := _parameterCnt + 1;
END_IF


// Check payload remaining ? 
IF ( ResponseData.IsPayloadRemaining)
THEN
  // Get Response.InProgress
 _response.InProgress := ResponseData.GetBool();
  // inc parameter counter
 _parameterCnt := _parameterCnt + 1;
END_IF


FOR _idx := 0 TO RobotLibraryParameter.SUB_PROGRAM_DATA_MAX
DO  
  // Check payload remaining ? 
  IF ( ResponseData.IsPayloadRemaining)
  THEN
    // Get Response.InProgress
   _response.ReturnData[_idx] := ResponseData.GetByte();  
    // inc parameter counter
   _parameterCnt := _parameterCnt + 1;
  END_IF   
END_FOR

// Create logging
ParseResponsePayloadLog(ResponseData := ResponseData, Timestamp := Timestamp, ParameterCnt := _parameterCnt);
                
END_METHOD

METHOD INTERNAL ParseResponsePayloadLog
VAR_INPUT
  /// Response data
  ResponseData : RobotLibraryResponseDataFB;
  /// Timestamp
  Timestamp    : SystemTime;  
  /// Parameter count
  ParameterCnt : DINT;
END_VAR
VAR
  /// internal index for loops
 _idx : DINT;
END_VAR
                  // Create log entry for Parameter start
CreateLogMessagePara1 ( Timestamp   := Timestamp,
                        MessageType := MessageType.CMD,
                        Severity    := Severity.DEBUG,
                        MessageCode := 0,
                        MessageText := '{1} parameter(s) to parse from the response data:',
                        Para1       := DINT_TO_STRING(ParameterCnt));
                        

// Return if no parameter is remaining...
IF ( ParameterCnt = 0 ) THEN RETURN; END_IF
// dec remaining parameter(s)                        
ParameterCnt := ParameterCnt - 1;
// Create log entry for InvocationCounter
CreateLogMessagePara1 ( Timestamp   := Timestamp,
                        MessageType := MessageType.CMD,
                        Severity    := Severity.DEBUG,
                        MessageCode := 0,
                        MessageText := 'Response.InvocationCounter = {1}',
                        Para1       :=  USINT_TO_STRING(_response.InvocationCounter));


// Return if no parameter is remaining...
IF ( ParameterCnt = 0 ) THEN RETURN; END_IF
// dec remaining parameter(s)                        
ParameterCnt := ParameterCnt - 1;
// Create log entry for Reserve
CreateLogMessagePara1 ( Timestamp   := Timestamp,
                        MessageType := MessageType.CMD,
                        Severity    := Severity.DEBUG,
                        MessageCode := 0,
                        MessageText := 'Response.Reserve = {1}',
                        Para1       :=  SINT_TO_STRING(_response.Reserve));


// Return if no parameter is remaining...
IF ( ParameterCnt = 0 ) THEN RETURN; END_IF
// dec remaining parameter(s)                        
ParameterCnt := ParameterCnt - 1;
// Create log entry for OriginID
CreateLogMessagePara1 ( Timestamp   := Timestamp,
                        MessageType := MessageType.CMD,
                        Severity    := Severity.DEBUG,
                        MessageCode := 0,
                        MessageText := 'Response.OriginID = {1}',
                        Para1       :=  INT_TO_STRING(_response.OriginID));


// Return if no parameter is remaining...
IF ( ParameterCnt = 0 ) THEN RETURN; END_IF
// dec remaining parameter(s)                        
ParameterCnt := ParameterCnt - 1;
// Create log entry for Progress
CreateLogMessagePara1 ( Timestamp   := Timestamp,
                        MessageType := MessageType.CMD,
                        Severity    := Severity.DEBUG,
                        MessageCode := 0,
                        MessageText := 'Response.Progress = {1}',
                        Para1       :=  UINT_TO_STRING(_response.Progress));


// Return if no parameter is remaining...
IF ( ParameterCnt = 0 ) THEN RETURN; END_IF
// dec remaining parameter(s)                        
ParameterCnt := ParameterCnt - 1;
// Create log entry for InProgress
CreateLogMessagePara1 ( Timestamp   := Timestamp,
                        MessageType := MessageType.CMD,
                        Severity    := Severity.DEBUG,
                        MessageCode := 0,
                        MessageText := 'Response.InProgress = {1}',
                        Para1       :=  BOOL_TO_STRING(_response.InProgress));


// Return if no parameter is remaining...
IF ( ParameterCnt = 0 ) THEN RETURN; END_IF
// dec remaining parameter(s)                        
ParameterCnt := ParameterCnt - 1;
// Create log entry for ReturnData[x]
FOR _idx := 0 TO RobotLibraryParameter.SUB_PROGRAM_DATA_MAX
DO
  CreateLogMessagePara2 ( Timestamp   := Timestamp,
                          MessageType := MessageType.CMD,
                          Severity    := Severity.DEBUG,
                          MessageCode := 0,
                          MessageText := 'Response.ReturnData[{2}] = {1}',
                          Para1       :=  BYTE_TO_STRING(_response.ReturnData[_idx]),
                          Para2       :=  DINT_TO_STRING(_idx));
END_FOR
                
END_METHOD

METHOD PROTECTED Reset : DINT
VAR_INPUT
END_VAR
                  Reset := SUPER^.Reset();

Done               := FALSE;
Busy               := FALSE;

Valid              := FALSE;
InProgress         := FALSE;
CommandAborted     := FALSE;
ParameterAccepted  := FALSE;

CommandBuffered    := FALSE;
CommandAborted     := FALSE;
CommandInterrupted := FALSE; 
                
END_METHOD
END_FUNCTION_BLOCK

/// Turn on/off the collision detection
FUNCTION_BLOCK MC_CollisionDetectionFB EXTENDS RobotLibraryBaseExecuteFB
// ------------------------------------------------------------------------- 
//  SRCI Robot Library                                                
// ------------------------------------------------------------------------- 
//                                                                           
//  Object:      CollisionDetectionFB                                       
//  Author:      Thorsten Brach                                                
//  Date:        2024-06-01
//
//  Description:                                              
//   
//                                                                           
//  Copyright: 
//    (C) 2024 Thorsten Brach. All rights reserved                                                                                                                                            
//             Licensed under the MIT License.
//                                                                           
//  Disclaimer:                                                                           
//    This project is provided without any guarantee and can be used for   
//    private and commercial purposes. Any use is at the user’s 
//    own risk and responsibility.
//
// -------------------------------------------------------------------------
VAR_INPUT
  /// Processing mode
  ProcessingMode     : ProcessingMode;
  /// Defines the target sequence in which the command will be executed
  SequenceFlag       : SequenceFlag; 
  /// Command parameter 
  ParCmd             : CollisionDetectionParCmd;
END_VAR
VAR_OUTPUT
  /// Command is transferred and confirmed by the RC
  CommandBuffered    : BOOL;
  /// The command was aborted by another command.
  CommandAborted     : BOOL;
  /// TRUE, while command is interrupted during execution and can be continued
  CommandInterrupted : BOOL;  
  /// command results
  OutCmd             : CollisionDetectionOutCmd;      
END_VAR

VAR
  /// internal copy of command parameter 
 _parCmd             : CollisionDetectionParCmd;
  /// command data to send
 _command            : CollisionDetectionSendData;
  /// response data received
 _response           : CollisionDetectionRecvData;      
END_VAR

            SUPER^(AxesGroup := AxesGroup);
          

METHOD INTERNAL CheckAddParameter : BOOL
VAR_INPUT
  /// Payload pointer
  PayloadPtr : UDINT;
END_VAR
VAR
  /// Payload as byte array
  Payload    : ARRAY [1..SIZEOF(_command)] OF BYTE;
  /// Null Byte array 
  Null       : ARRAY [1..SIZEOF(_command)] OF BYTE;
  /// Data length to compare
  DataLen    : UDINT;
END_VAR
                  // Payload pointer must be decreased by one byte, because ADR(Payload) is already one byte !
PayloadPtr := LIMIT (0, PayloadPtr - 1, SIZEOF(Payload) -1);
// Convert command struct to payload array
SysDepMemCpy( pDest := ADR(Payload), pSrc := ADR(_command), DataLen := SIZEOF(_command));
// Calculate the data length to compare - at least one byte must be compared !
DataLen := LIMIT(1, SIZEOF(Payload) - PayloadPtr, SIZEOF(Payload)); 
// Compare Payload-Array with Null-Byte-Array
CheckAddParameter := SysDepMemCmp( pData1 := ADR(Payload) + PayloadPtr , pData2 := ADR(Null), DataLen := DataLen) <>  RobotLibraryConstants.OK ;
                
END_METHOD

METHOD PROTECTED CheckFunctionSupported : BOOL
VAR_IN_OUT
  /// Robot assignment of function
  AxesGroup : AxesGroup; 
END_VAR
                  CheckFunctionSupported := AxesGroup.State.RobotData.RCSupportedFunctions.CollisionDetection;

IF ( NOT CheckFunctionSupported )
THEN
  // call base implementation for set error and create log entry
  SUPER^.CheckFunctionSupported(AxesGroup := AxesGroup);
END_IF
                
END_METHOD

METHOD PROTECTED CheckParameterChanged : BOOL
VAR_IN_OUT
  /// Robot assignment of function
  AxesGroup    : AxesGroup; 
END_VAR
                  // Check ParCmd Size is > 0, because MemCmp does not work correctly with size = 0
IF (SIZEOF(ParCmd) = 0) OR (_stepCmd = 0)
THEN 
  RETURN;
END_IF

// compare memory 
_parameterChanged := ( SysDepMemCmp(pData1 := ADR(ParCmd), pData2 := ADR(_parCmd), DataLen := SIZEOF(ParCmd)) <> RobotLibraryConstants.OK );

// check parameter valid ?
_parameterValid   := CheckParameterValid( AxesGroup := AxesGroup );

IF ((  _parameterChanged        )  AND 
    (  _parameterValid          )) OR
    (  _parameterUpdateInternal )  
THEN  
  // Create log entry for parameter changed event
  CreateLogMessagePara1 ( Timestamp   := AxesGroup.State.SystemTime,
                          MessageType := MessageType.CMD,
                          Severity    := Severity.DEBUG,
                          MessageCode := 0,
                          MessageText := 'NotifyParameterChanged Event {1}',
                          Para1       :=  '' );

  // reset internal flag for send parameter update
 _parameterUpdateInternal := FALSE;
  // update internal copy of parameters 
 _parCmd := ParCmd;
  // inc parameter sequence
 _command.ParSeq := _command.ParSeq + 1;
  // update command data  
  CommandData := CreateCommandPayload(AxesGroup := AxesGroup); // ( Access via reference to rCommandFB in ACR )
  // notify active command register 
  AxesGroup.Acyclic.ActiveCommandRegister.NotifyParameterChanged := _uniqueID;
END_IF
                
END_METHOD

METHOD PROTECTED CheckParameterValid : BOOL
VAR_IN_OUT
  /// Robot assignment of function
  AxesGroup : AxesGroup; 
END_VAR

VAR
  /// internal index for loops
 _idx : DINT;
END_VAR
                  CheckParameterValid := TRUE;

// Check ParCmd.ProcessingMode defined ? 
IF (( ProcessingMode < ProcessingModeEnum.BUFFERED         ) AND
    ( ProcessingMode > ProcessingModeEnum.TRIGGER_MULTIPLE ))
THEN
  // Parameter not valid
  CheckParameterValid := FALSE;
  // Set error
  SetError( ErrorID := RobotLibraryErrorIdEnum.ERR_PROCESSINGMODE_NOT_DEFINED, Overwrite := TRUE );
  // Create log entry
  CreateLogMessagePara1 ( Timestamp   := AxesGroup.State.SystemTime,
                          MessageType := MessageType.CMD,
                          Severity    := Severity.ERROR,
                          MessageCode := ErrorID,
                          MessageText := 'Invalid Parameter ParCmd.ProcessingMode = {1}',
                          Para1       := PROCESSING_MODE_TO_STRING(ProcessingMode));
  RETURN;                          
END_IF

// Check ProcessingMode valid ? 
IF (( ProcessingMode <> ProcessingModeEnum.BUFFERED ) AND
    ( ProcessingMode <> ProcessingModeEnum.ABORTING ) AND  
    ( ProcessingMode <> ProcessingModeEnum.PARALLEL ))
THEN
  // Parameter not valid
  CheckParameterValid := FALSE;
  // Set error
  SetError( ErrorID := RobotLibraryErrorIdEnum.ERR_PROCESSINGMODE_NOT_ALLOWED, Overwrite := TRUE );
  // Create log entry
  CreateLogMessagePara1 ( Timestamp   := AxesGroup.State.SystemTime,
                          MessageType := MessageType.CMD,
                          Severity    := Severity.ERROR,
                          MessageCode := ErrorID,
                          MessageText := 'Invalid Parameter ProcessingMode = {1}',
                          Para1       := PROCESSING_MODE_TO_STRING(ProcessingMode));
  RETURN;                          
END_IF

// Check SequenceFlag valid ? 
IF (( SequenceFlag <> SequenceFlagEnum.PRIMARY_SEQUENCE   ) AND
    ( SequenceFlag <> SequenceFlagEnum.SECONDARY_SEQUENCE ))
THEN
  // Parameter not valid
  CheckParameterValid := FALSE;
  // Set error
  SetError( ErrorID := RobotLibraryErrorIdEnum.ERR_SEQFLAG_NOT_ALLOWED, Overwrite := TRUE );
  // Create log entry
  CreateLogMessagePara1 ( Timestamp   := AxesGroup.State.SystemTime,
                          MessageType := MessageType.CMD,
                          Severity    := Severity.ERROR,
                          MessageCode := ErrorID,
                          MessageText := 'Invalid Parameter SequenceFlag = {1}',
                          Para1       := SEQUENCE_FLAG_TO_STRING(SequenceFlag));
  RETURN;                          
END_IF


// Check ParCmd.ReactionMode valid ? 
IF (( ParCmd.ReactionMode < CollisionReactionMode.STANDING_STILL    ) OR  
    ( ParCmd.ReactionMode > CollisionReactionMode.REVERSED_MOVEMENT ))
THEN
  // Parameter not valid
  CheckParameterValid := FALSE;
  // Set error
  SetError( ErrorID := RobotLibraryErrorIdEnum.ERR_INVALID_PAR_CMD, Overwrite := TRUE ); 
  // Create log entry
  CreateLogMessagePara1 ( Timestamp   := AxesGroup.State.SystemTime,
                          MessageType := MessageType.CMD,
                          Severity    := Severity.ERROR,
                          MessageCode := ErrorID,
                          MessageText := 'Invalid Parameter ParCmd.ReactionMode = {1}',
                          Para1       :=  COLLISION_REACTION_MODE_TO_STRING(ParCmd.ReactionMode));
  RETURN;                          
END_IF


// Check ParCmd.ThresholdMode valid ? 
IF (( ParCmd.ThresholdMode <> ThresholdMode.AUTOMATIC ) AND  
    ( ParCmd.ThresholdMode <> ThresholdMode.MANUAL    ))
THEN
  // Parameter not valid
  CheckParameterValid := FALSE;
  // Set error
  SetError( ErrorID := RobotLibraryErrorIdEnum.ERR_INVALID_PAR_CMD, Overwrite := TRUE );
  // Create log entry
  CreateLogMessagePara1 ( Timestamp   := AxesGroup.State.SystemTime,
                          MessageType := MessageType.CMD,
                          Severity    := Severity.ERROR,
                          MessageCode := ErrorID,
                          MessageText := 'Invalid Parameter ParCmd.ThresholdMode = {1}',
                          Para1       := THRESHOLD_MODE_TO_STRING(ParCmd.ThresholdMode));
  RETURN;                          
END_IF



// Check ParCmd.Sensitivity valid ? 
IF (( SysDepIsValidReal(ParCmd.Sensitivity) = FALSE ) OR
    ( ParCmd.Sensitivity                    <     0 ) OR  
    ( ParCmd.Sensitivity                    >   200 ))
THEN
  // Parameter not valid
  CheckParameterValid := FALSE;
  // Set error
  SetError( ErrorID := RobotLibraryErrorIdEnum.ERR_INVALID_PAR_CMD, Overwrite := TRUE );
  
  // Create log entry
  CreateLogMessagePara1 ( Timestamp   := AxesGroup.State.SystemTime,
                          MessageType := MessageType.CMD,
                          Severity    := Severity.ERROR,
                          MessageCode := ErrorID,
                          MessageText := 'Invalid Parameter ParCmd.Sensitivity = {1}',
                          Para1       := VALID_REAL_TO_STRING(ParCmd.Sensitivity));
  RETURN;                          
END_IF



FOR _idx := 0 TO 6
DO
  // Check ParCmd.SensitivityAxis valid ? 
  IF (( SysDepIsValidReal(ParCmd.SensitivityAxis[_idx]) = FALSE ) OR
      (                   ParCmd.SensitivityAxis[_idx]  <     0 ) OR  
      (                   ParCmd.SensitivityAxis[_idx]  >   200 ))      
  THEN
    // Parameter not valid
    CheckParameterValid := FALSE;
    // Set error
    SetError( ErrorID := RobotLibraryErrorIdEnum.ERR_INVALID_PAR_CMD, Overwrite := TRUE ); 
    // Create log entry
    CreateLogMessagePara2 ( Timestamp   := AxesGroup.State.SystemTime,
                            MessageType := MessageType.CMD,
                            Severity    := Severity.ERROR,
                            MessageCode := ErrorID,
                            MessageText := 'Invalid Parameter ParCmd.SensitivityAxis[{2}] = {1}',
                            Para1       := VALID_REAL_TO_STRING(ParCmd.SensitivityAxis[_idx]),
                            Para2       := DINT_TO_STRING(_idx));
    EXIT;
    RETURN;                          
  END_IF
END_FOR  


FOR _idx := 0 TO 6
DO
  // Check ParCmd.LimitAxis valid ? 
  IF (( SysDepIsValidReal(ParCmd.LimitAxis[_idx]) = FALSE ))
  THEN
    // Parameter not valid
    CheckParameterValid := FALSE;
    // Set error
    SetError( ErrorID := RobotLibraryErrorIdEnum.ERR_INVALID_PAR_CMD, Overwrite := TRUE ); 
    // Create log entry
    CreateLogMessagePara2 ( Timestamp   := AxesGroup.State.SystemTime,
                            MessageType := MessageType.CMD,
                            Severity    := Severity.ERROR,
                            MessageCode := ErrorID,
                            MessageText := 'Invalid Parameter ParCmd.LimitAxis[{2}] = {1}',
                            Para1       := VALID_REAL_TO_STRING(ParCmd.LimitAxis[_idx]),
                            Para2       := DINT_TO_STRING(_idx));
    EXIT;
    RETURN;                          
  END_IF
END_FOR  


// Check ParCmd.UnitLimitAxis valid ? 
IF (( ParCmd.UnitLimitAxis <> UnitLimitAxis.PERCENTAGE  ) AND  
    ( ParCmd.UnitLimitAxis <> UnitLimitAxis.NEWTONMETER ) AND
    ( ParCmd.UnitLimitAxis <> UnitLimitAxis.MILLIAMPERE ))
THEN
  // Parameter not valid
  CheckParameterValid := FALSE;
  // Set error
  SetError( ErrorID := RobotLibraryErrorIdEnum.ERR_INVALID_PAR_CMD, Overwrite := TRUE );
  // Create log entry
  CreateLogMessagePara1 ( Timestamp   := AxesGroup.State.SystemTime,
                          MessageType := MessageType.CMD,
                          Severity    := Severity.ERROR,
                          MessageCode := ErrorID,
                          MessageText := 'Invalid Parameter ParCmd.UnitLimitAxis = {1}',
                          Para1       := THRESHOLD_MODE_TO_STRING(ParCmd.UnitLimitAxis));
  RETURN;                          
END_IF
                
END_METHOD

METHOD INTERNAL CreateCommandPayload : RobotLibraryCommandDataFB
VAR_IN_OUT
  /// Robot assignment of function
  AxesGroup : AxesGroup; 
END_VAR
VAR
  /// Parameter count
 _parameterCnt : DINT;
  /// internal index for loops
 _idx          : DINT;
END_VAR
// Table 6-790: Sent CMD payload (PLC to RC) of "CollisionDetection"
// --------------------------
// Header
// --------------------------
// Byte 00 : UINT  - Type HB     
// Byte 01 :       - Type LB    
// Byte 02 : USINT - Reserve | ExecutionMode
// Byte 03 : USINT - ParSeq  | Priority
// --------------------------
// Datablock
// --------------------------
// Byte 04 : BOOL      - ActivateMonitoring
// Byte 05 : USINT     - UnitLimitAxis
// Byte 06 : USINT     - ThresholdMode
// Byte 07 : USINT     - ReactionMode
// Byte 08 : INT       - Sensitivity
// Byte 09 :           - Reserved
// Byte 10 : INT       - SensitivityAxis[0]
// Byte 11 :           - Reserved
// Byte 12 : INT       - SensitivityAxis[1]
// Byte 13 :           - Reserved
// Byte 14 : INT       - SensitivityAxis[2]
// Byte 15 :           - Reserved
// Byte 16 : INT       - SensitivityAxis[3]
// Byte 17 :           - Reserved
// Byte 18 : INT       - SensitivityAxis[4]
// Byte 19 :           - Reserved
// Byte 20 : INT       - SensitivityAxis[5]
// Byte 21 :           - Reserved
// Byte 22 : INT       - SensitivityAxis[6]
// Byte 23 :           - Reserved
// Byte 24 : REAL      - LimitAxis[0] HW HB
// Byte 25 :           - LimitAxis[0] HW LB
// Byte 26 :           - LimitAxis[0] LW HB
// Byte 27 :           - LimitAxis[0] LW LB
// Byte 28 : REAL      - LimitAxis[1] HW HB
// Byte 29 :           - LimitAxis[1] HW LB
// Byte 30 :           - LimitAxis[1] LW HB
// Byte 31 :           - LimitAxis[1] LW LB
// Byte 32 : REAL      - LimitAxis[2] HW HB
// Byte 33 :           - LimitAxis[2] HW LB
// Byte 34 :           - LimitAxis[2] LW HB
// Byte 35 :           - LimitAxis[2] LW LB
// Byte 36 : REAL      - LimitAxis[3] HW HB
// Byte 37 :           - LimitAxis[3] HW LB
// Byte 38 :           - LimitAxis[3] LW HB
// Byte 39 :           - LimitAxis[3] LW LB
// Byte 40 : REAL      - LimitAxis[4] HW HB
// Byte 41 :           - LimitAxis[4] HW LB
// Byte 42 :           - LimitAxis[4] LW HB
// Byte 43 :           - LimitAxis[4] LW LB
// Byte 44 : REAL      - LimitAxis[5] HW HB
// Byte 45 :           - LimitAxis[5] HW LB
// Byte 46 :           - LimitAxis[5] LW HB
// Byte 47 :           - LimitAxis[5] LW LB
// Byte 48 : REAL      - LimitAxis[6] HW HB
// Byte 49 :           - LimitAxis[6] HW LB
// Byte 50 :           - LimitAxis[6] LW HB
// Byte 51 :           - LimitAxis[6] LW LB
// --------------------------
                  // set command parameter 
_command.CmdTyp               :=  CmdType.CollisionDetection;
_command.ExecMode             :=  ExecMode;
_command.ParSeq               := _command.ParSeq;
_command.Priority             :=  Priority;

_command.ActivateMonitoring   := _parCmd.ActivateMonitoring;
_command.UnitLimitAxis        := _parCmd.UnitLimitAxis;
_command.ThresholdMode        := _parCmd.ThresholdMode;
_command.ReactionMode         := _parCmd.ReactionMode;
_command.Sensitivity          :=  REAL_TO_PERCENT_INT(_parCmd.Sensitivity        , IsOptional := TRUE);
_command.SensitivityAxis[0]   :=  REAL_TO_PERCENT_INT(_parCmd.SensitivityAxis[0] , IsOptional := TRUE);
_command.SensitivityAxis[1]   :=  REAL_TO_PERCENT_INT(_parCmd.SensitivityAxis[1] , IsOptional := TRUE);
_command.SensitivityAxis[2]   :=  REAL_TO_PERCENT_INT(_parCmd.SensitivityAxis[2] , IsOptional := TRUE);
_command.SensitivityAxis[3]   :=  REAL_TO_PERCENT_INT(_parCmd.SensitivityAxis[3] , IsOptional := TRUE);
_command.SensitivityAxis[4]   :=  REAL_TO_PERCENT_INT(_parCmd.SensitivityAxis[4] , IsOptional := TRUE);
_command.SensitivityAxis[5]   :=  REAL_TO_PERCENT_INT(_parCmd.SensitivityAxis[5] , IsOptional := TRUE);
_command.SensitivityAxis[6]   :=  REAL_TO_PERCENT_INT(_parCmd.SensitivityAxis[6] , IsOptional := TRUE);
_command.LimitAxis[0]         := _parCmd.LimitAxis[0];
_command.LimitAxis[1]         := _parCmd.LimitAxis[1];
_command.LimitAxis[2]         := _parCmd.LimitAxis[2];
_command.LimitAxis[3]         := _parCmd.LimitAxis[3];
_command.LimitAxis[4]         := _parCmd.LimitAxis[4];
_command.LimitAxis[5]         := _parCmd.LimitAxis[5];
_command.LimitAxis[6]         := _parCmd.LimitAxis[6];



// copy command data to header
_cmdHeader := _command;
// call base implementation to copy header to payload buffer
CreateCommandPayload := SUPER^.CreateCommandPayload(AxesGroup := AxesGroup);


// Check parameter must be added ? 
IF ( CheckAddParameter(CreateCommandPayload.PayloadPtr))
THEN
  // add command.ActivateMonitoring
  CreateCommandPayload.AddBool(_command.ActivateMonitoring);
  // inc parameter counter
 _parameterCnt := _parameterCnt + 1;  
END_IF


// Check parameter must be added ? 
IF ( CheckAddParameter(CreateCommandPayload.PayloadPtr))
THEN
  // add command.UnitLimitAxis
  CreateCommandPayload.AddUsint(_command.UnitLimitAxis);
  // inc parameter counter
 _parameterCnt := _parameterCnt + 1;  
END_IF


// Check parameter must be added ? 
IF ( CheckAddParameter(CreateCommandPayload.PayloadPtr))
THEN
  // add command.ThresholdMode
  CreateCommandPayload.AddUsint(_command.ThresholdMode);
  // inc parameter counter
 _parameterCnt := _parameterCnt + 1;  
END_IF


// Check parameter must be added ? 
IF ( CheckAddParameter(CreateCommandPayload.PayloadPtr))
THEN
  // add command.ReactionMode
  CreateCommandPayload.AddUsint(_command.ReactionMode);
  // inc parameter counter
 _parameterCnt := _parameterCnt + 1;  
END_IF


// Check parameter must be added ? 
IF ( CheckAddParameter(CreateCommandPayload.PayloadPtr))
THEN
  // add command.Sensitivity
  CreateCommandPayload.AddInt(_command.Sensitivity);
  // inc parameter counter
 _parameterCnt := _parameterCnt + 1;  
END_IF


FOR _idx := 0 TO 6
DO
  // Check parameter must be added ? 
  IF ( CheckAddParameter(CreateCommandPayload.PayloadPtr))
  THEN
    // add command.SensitivityAxis[x]
    CreateCommandPayload.AddInt(_command.SensitivityAxis[_idx]);
    // inc parameter counter
   _parameterCnt := _parameterCnt + 1;  
  END_IF
END_FOR


FOR _idx := 0 TO 6
DO
  // Check parameter must be added ? 
  IF ( CheckAddParameter(CreateCommandPayload.PayloadPtr))
  THEN
    // add command.LimitAxis[x]
    CreateCommandPayload.AddReal(_command.LimitAxis[_idx]);
    // inc parameter counter
   _parameterCnt := _parameterCnt + 1;  
  END_IF
END_FOR


// Create logging
CreateCommandPayloadLog(AxesGroup := AxesGroup, ParameterCnt := _parameterCnt);
                
END_METHOD

METHOD INTERNAL CreateCommandPayloadLog
VAR_IN_OUT
  /// Robot assignment of function
  AxesGroup : AxesGroup; 
END_VAR
VAR_INPUT
  /// Parameter count
  ParameterCnt : DINT;
END_VAR
                  // Create log entry for Parameter start
CreateLogMessagePara1 ( Timestamp   := AxesGroup.State.SystemTime,
                        MessageType := MessageType.CMD,
                        Severity    := Severity.DEBUG,
                        MessageCode := 0,
                        MessageText := 'Create command payload with {1} parameter(s) :',
                        Para1       := DINT_TO_STRING(ParameterCnt));
  

// Return if no parameter is remaining...
IF ( ParameterCnt = 0 ) THEN RETURN; END_IF
// dec remaining parameter(s)                        
ParameterCnt := ParameterCnt - 1;
// Create log entry for ActivateMonitoring
CreateLogMessagePara1 ( Timestamp   := AxesGroup.State.SystemTime,
                        MessageType := MessageType.CMD,
                        Severity    := Severity.DEBUG,
                        MessageCode := 0,
                        MessageText := 'Command.ActivateMonitoring = {1}',
                        Para1       :=  BOOL_TO_STRING(_command.ActivateMonitoring));


// Return if no parameter is remaining...
IF ( ParameterCnt = 0 ) THEN RETURN; END_IF
// dec remaining parameter(s)                        
ParameterCnt := ParameterCnt - 1;
// Create log entry for UnitLimitAxis
CreateLogMessagePara1 ( Timestamp   := AxesGroup.State.SystemTime,
                        MessageType := MessageType.CMD,
                        Severity    := Severity.DEBUG,
                        MessageCode := 0,
                        MessageText := 'Command.UnitLimitAxis = {1}',
                        Para1       :=  USINT_TO_STRING(_command.UnitLimitAxis));


// Return if no parameter is remaining...
IF ( ParameterCnt = 0 ) THEN RETURN; END_IF
// dec remaining parameter(s)                        
ParameterCnt := ParameterCnt - 1;
// Create log entry for ThresholdMode
CreateLogMessagePara1 ( Timestamp   := AxesGroup.State.SystemTime,
                        MessageType := MessageType.CMD,
                        Severity    := Severity.DEBUG,
                        MessageCode := 0,
                        MessageText := 'Command.ThresholdMode = {1}',
                        Para1       :=  THRESHOLD_MODE_TO_STRING(_command.ThresholdMode)); 


// Return if no parameter is remaining...
IF ( ParameterCnt = 0 ) THEN RETURN; END_IF
// dec remaining parameter(s)                        
ParameterCnt := ParameterCnt - 1;
// Create log entry for ReactionMode
CreateLogMessagePara1 ( Timestamp   := AxesGroup.State.SystemTime,
                        MessageType := MessageType.CMD,
                        Severity    := Severity.DEBUG,
                        MessageCode := 0,
                        MessageText := 'Command.ReactionMode = {1}',
                        Para1       :=  COLLISION_REACTION_MODE_TO_STRING(_command.ReactionMode)); 


// Return if no parameter is remaining...
IF ( ParameterCnt = 0 ) THEN RETURN; END_IF
// dec remaining parameter(s)                        
ParameterCnt := ParameterCnt - 1;
// Create log entry for Sensitivity
CreateLogMessagePara1 ( Timestamp   := AxesGroup.State.SystemTime,
                        MessageType := MessageType.CMD,
                        Severity    := Severity.DEBUG,
                        MessageCode := 0,
                        MessageText := 'Command.Sensitivity = {1}',
                        Para1       :=  INT_TO_STRING(_command.Sensitivity)); 


// Return if no parameter is remaining...
IF ( ParameterCnt = 0 ) THEN RETURN; END_IF
// dec remaining parameter(s)                        
ParameterCnt := ParameterCnt - 1;
// Create log entry for SensitivityAxis[1]
CreateLogMessagePara1 ( Timestamp   := AxesGroup.State.SystemTime,
                        MessageType := MessageType.CMD,
                        Severity    := Severity.DEBUG,
                        MessageCode := 0,
                        MessageText := 'Command.SensitivityAxis[1] = {1}',
                        Para1       :=  INT_TO_STRING(_command.SensitivityAxis[1]));
 

// Return if no parameter is remaining...
IF ( ParameterCnt = 0 ) THEN RETURN; END_IF
// dec remaining parameter(s)                        
ParameterCnt := ParameterCnt - 1;
// Create log entry for SensitivityAxis[2]
CreateLogMessagePara1 ( Timestamp   := AxesGroup.State.SystemTime,
                        MessageType := MessageType.CMD,
                        Severity    := Severity.DEBUG,
                        MessageCode := 0,
                        MessageText := 'Command.SensitivityAxis[2] = {1}',
                        Para1       :=  INT_TO_STRING(_command.SensitivityAxis[2]));
                        

// Return if no parameter is remaining...
IF ( ParameterCnt = 0 ) THEN RETURN; END_IF
// dec remaining parameter(s)                        
ParameterCnt := ParameterCnt - 1;
// Create log entry for SensitivityAxis[3]
CreateLogMessagePara1 ( Timestamp   := AxesGroup.State.SystemTime,
                        MessageType := MessageType.CMD,
                        Severity    := Severity.DEBUG,
                        MessageCode := 0,
                        MessageText := 'Command.SensitivityAxis[3] = {1}',
                        Para1       :=  INT_TO_STRING(_command.SensitivityAxis[3]));
                        

// Return if no parameter is remaining...
IF ( ParameterCnt = 0 ) THEN RETURN; END_IF
// dec remaining parameter(s)                        
ParameterCnt := ParameterCnt - 1;
// Create log entry for SensitivityAxis[4]
CreateLogMessagePara1 ( Timestamp   := AxesGroup.State.SystemTime,
                        MessageType := MessageType.CMD,
                        Severity    := Severity.DEBUG,
                        MessageCode := 0,
                        MessageText := 'Command.SensitivityAxis[4] = {1}',
                        Para1       :=  INT_TO_STRING(_command.SensitivityAxis[4])); 
 

// Return if no parameter is remaining...
IF ( ParameterCnt = 0 ) THEN RETURN; END_IF
// dec remaining parameter(s)                        
ParameterCnt := ParameterCnt - 1;
// Create log entry for SensitivityAxis[5]
CreateLogMessagePara1 ( Timestamp   := AxesGroup.State.SystemTime,
                        MessageType := MessageType.CMD,
                        Severity    := Severity.DEBUG,
                        MessageCode := 0,
                        MessageText := 'Command.SensitivityAxis[5] = {1}',
                        Para1       :=  INT_TO_STRING(_command.SensitivityAxis[5]));


// Return if no parameter is remaining...
IF ( ParameterCnt = 0 ) THEN RETURN; END_IF
// dec remaining parameter(s)                        
ParameterCnt := ParameterCnt - 1;
// Create log entry for SensitivityAxis[6]
CreateLogMessagePara1 ( Timestamp   := AxesGroup.State.SystemTime,
                        MessageType := MessageType.CMD,
                        Severity    := Severity.DEBUG,
                        MessageCode := 0,
                        MessageText := 'Command.SensitivityAxis[6] = {1}',
                        Para1       :=  INT_TO_STRING(_command.SensitivityAxis[6]));
                        

// Return if no parameter is remaining...
IF ( ParameterCnt = 0 ) THEN RETURN; END_IF
// dec remaining parameter(s)                        
ParameterCnt := ParameterCnt - 1;
// Create log entry for LimitAxis[1]
CreateLogMessagePara1 ( Timestamp   := AxesGroup.State.SystemTime,
                        MessageType := MessageType.CMD,
                        Severity    := Severity.DEBUG,
                        MessageCode := 0,
                        MessageText := 'Command.LimitAxis[1] = {1}',
                        Para1       :=  REAL_TO_STRING(_command.LimitAxis[1]));


// Return if no parameter is remaining...
IF ( ParameterCnt = 0 ) THEN RETURN; END_IF
// dec remaining parameter(s)                        
ParameterCnt := ParameterCnt - 1;
// Create log entry for LimitAxis[2]
CreateLogMessagePara1 ( Timestamp   := AxesGroup.State.SystemTime,
                        MessageType := MessageType.CMD,
                        Severity    := Severity.DEBUG,
                        MessageCode := 0,
                        MessageText := 'Command.LimitAxis[2] = {1}',
                        Para1       :=  REAL_TO_STRING(_command.LimitAxis[2]));
                        

// Return if no parameter is remaining...
IF ( ParameterCnt = 0 ) THEN RETURN; END_IF
// dec remaining parameter(s)                        
ParameterCnt := ParameterCnt - 1;
// Create log entry for LimitAxis[3]
CreateLogMessagePara1 ( Timestamp   := AxesGroup.State.SystemTime,
                        MessageType := MessageType.CMD,
                        Severity    := Severity.DEBUG,
                        MessageCode := 0,
                        MessageText := 'Command.LimitAxis[3] = {1}',
                        Para1       :=  REAL_TO_STRING(_command.LimitAxis[3]));
                        

// Return if no parameter is remaining...
IF ( ParameterCnt = 0 ) THEN RETURN; END_IF
// dec remaining parameter(s)                        
ParameterCnt := ParameterCnt - 1;
// Create log entry for LimitAxis[4]
CreateLogMessagePara1 ( Timestamp   := AxesGroup.State.SystemTime,
                        MessageType := MessageType.CMD,
                        Severity    := Severity.DEBUG,
                        MessageCode := 0,
                        MessageText := 'Command.LimitAxis[4] = {1}',
                        Para1       :=  REAL_TO_STRING(_command.LimitAxis[4]));


// Return if no parameter is remaining...
IF ( ParameterCnt = 0 ) THEN RETURN; END_IF
// dec remaining parameter(s)                        
ParameterCnt := ParameterCnt - 1;
// Create log entry for LimitAxis[5]
CreateLogMessagePara1 ( Timestamp   := AxesGroup.State.SystemTime,
                        MessageType := MessageType.CMD,
                        Severity    := Severity.DEBUG,
                        MessageCode := 0,
                        MessageText := 'Command.LimitAxis[5] = {1}',
                        Para1       :=  REAL_TO_STRING(_command.LimitAxis[5]));


// Return if no parameter is remaining...
IF ( ParameterCnt = 0 ) THEN RETURN; END_IF
// dec remaining parameter(s)                        
ParameterCnt := ParameterCnt - 1;
// Create log entry for LimitAxis[6]
CreateLogMessagePara1 ( Timestamp   := AxesGroup.State.SystemTime,
                        MessageType := MessageType.CMD,
                        Severity    := Severity.DEBUG,
                        MessageCode := 0,
                        MessageText := 'Command.LimitAxis[6] = {1}',
                        Para1       :=  REAL_TO_STRING(_command.LimitAxis[6]));
                
END_METHOD

METHOD FB_init : BOOL
VAR_INPUT
  /// if TRUE, the retain variables are initialized (warm start / cold start)
  bInitRetains : BOOL; 
  /// if TRUE, the instance afterwards gets moved into the copy code (online change)
  bInCopyCode  : BOOL;  
END_VAR
                  MyType := 'MC_CollisionDetectionFB';

ExecMode       := ExecutionMode.PARALLEL;
Priority       := PriorityLevel.NORMAL;
ProcessingMode := ProcessingModeEnum.PARALLEL;
SequenceFlag   := SequenceFlagEnum.NO_SEQUENCE;  

                
END_METHOD

METHOD PROTECTED OnExecRun : DINT
VAR_IN_OUT
  /// Robot assignment of function
  AxesGroup : AxesGroup; 
END_VAR
                  // call base implementation
SUPER^.OnExecRun(AxesGroup := AxesGroup);

CASE _stepCmd OF
  
  00:  IF ( _execute_R.Q ) AND ( NOT Error) 
       THEN
         // Check function is supported and parameter are valid ?
         IF (( CheckFunctionSupported( AxesGroup := AxesGroup )) AND
             ( CheckParameterValid   ( AxesGroup := AxesGroup )))      
         THEN
           // set busy flag
           Busy := TRUE;
           // Reset command outputs
           SysDepMemSet(pDest := ADR(OutCmd), Value := 0, DataLen := SIZEOF(OutCmd));         
           // apply command parameter
          _parCmd := ParCmd;
           // init parameter sequence
          _command.ParSeq := 1;
           // create command data
           CommandData := CreateCommandPayload(AxesGroup := AxesGroup);
           // Add command to active command register
          _uniqueID := AxesGroup.Acyclic.ActiveCommandRegister.AddCmd( pCommandFB := ADR(THIS^ ));     
           // set timeout
           SetTimeout(PT := _timeoutCmd, rTimer := _timerCmd);
           // inc step counter
          _stepCmd := _stepCmd + 1; 
         END_IF
       END_IF
     

  01:  // Wait for responce received
       IF ( _responseReceived )
       THEN
         // reset response received flag
        _responseReceived := FALSE;
         // update state flags
         OnUpdateStateFlags(_response.State);
         // update state flags
         OnApplyOutCmd(_response.State);
               
         // Done, Aborted or Error ?
         IF (_response.State >= CmdMessageState.DONE )
         THEN
           // set timeout
           SetTimeout(PT := _timeoutCmd, rTimer := _timerCmd);
           // inc step counter
          _stepCmd := _stepCmd + 1; 
         END_IF
       END_IF

  02: IF ( NOT Execute)
      THEN
        Reset();
      END_IF     
ELSE
  // invalid step
  SetError( ErrorID := RobotLibraryErrorIdEnum.ERR_INVALID_STEP, Overwrite := TRUE );
END_CASE


// Reset FB
IF ( NOT Execute )
THEN
  Reset();
END_IF
                
END_METHOD

METHOD PROTECTED OnUpdateStateFlags
VAR_INPUT
  /// Command message state
  State : CmdMessageState;
END_VAR
                  // Reset State flags
CommandAborted     := FALSE;
CommandInterrupted := FALSE;
Done               := FALSE;

CASE State OF

  // No operation or process is active
  CmdMessageState.EMPTY               :;
  // Created but not yet started
  CmdMessageState.CREATED             :;
  // Buffered and awaiting execution
  CmdMessageState.BUFFERED            : CommandBuffered    := TRUE;
  // Buffered in planner for future execution
  CmdMessageState.BUFFERED_IN_PLANNER : CommandBuffered    := TRUE;
  // Currently active and in progress
  CmdMessageState.ACTIVE              :;
  // Interrupted and awaiting continuation
  CmdMessageState.INTERRUPTED         : CommandInterrupted := TRUE;
  // Requested for abort
  CmdMessageState.ABORT_REQUEST       :;
  // Successfully completed
  CmdMessageState.DONE                : Done               := TRUE;
                                        Busy               := FALSE;
  // Aborted before completion
  CmdMessageState.ABORTED             : CommandAborted     := TRUE;
                                        Busy               := FALSE;
  // Encountered an error during execution
  CmdMessageState.ERROR               : Error              := TRUE;
                                        Busy               := FALSE;
END_CASE
                
END_METHOD

METHOD INTERNAL ParseResponsePayload : DINT
VAR_INPUT
  /// Response data
  ResponseData : RobotLibraryResponseDataFB;
  /// Timestamp
  Timestamp    : SystemTime;  
END_VAR
VAR
  /// Parameter count
 _parameterCnt : DINT;
END_VAR
// Table 6-791: Received CMD payload (RC to PLC) of "CollisionDetection"
// --------------------------
// Header
// --------------------------
// Byte 00 : USINT - ParSeq | State     
// Byte 01 : SINT  - AlarmMessageSeverity    
// Byte 02 : UINT  - AlarmMessageCode HB
// Byte 03 :       - AlarmMessageCode LB
                  // call base implementation to parse the header from payload buffer
ResponseData.PayloadPtr := SUPER^.ParseResponsePayload(ResponseData := ResponseData, Timestamp := Timestamp);

// copy parsed header to response
_response.ParSeq               := _rspHeader.ParSeq;
_response.State                := _rspHeader.State;
_response.AlarmMessageSeverity := _rspHeader.AlarmMessageSeverity;
_response.AlarmMessageCode     := _rspHeader.AlarmMessageCode;

// Create logging
ParseResponsePayloadLog(ResponseData := ResponseData, Timestamp := Timestamp, ParameterCnt := _parameterCnt);
                
END_METHOD

METHOD INTERNAL ParseResponsePayloadLog
VAR_INPUT
  /// Response data
  ResponseData : RobotLibraryResponseDataFB;
  /// Timestamp
  Timestamp    : SystemTime;  
  /// Parameter count
  ParameterCnt : DINT;
END_VAR
                  // Create log entry for Parameter start
CreateLogMessagePara1 ( Timestamp   := Timestamp,
                        MessageType := MessageType.CMD,
                        Severity    := Severity.DEBUG,
                        MessageCode := 0,
                        MessageText := '{1} parameter(s) to parse from the response data:',
                        Para1       := DINT_TO_STRING(ParameterCnt));

                        
// Return if no parameter is remaining...
IF ( ParameterCnt = 0 ) THEN RETURN; END_IF
// dec remaining parameter(s)                        
ParameterCnt := ParameterCnt - 1;
// Create log entry for no parameter 
CreateLogMessage      ( Timestamp   := Timestamp,
                        MessageType := MessageType.CMD,
                        Severity    := Severity.DEBUG,
                        MessageCode := 0,
                        MessageText := 'This command has no parameter to parse...');
                
END_METHOD

METHOD PROTECTED Reset : DINT
VAR_INPUT
END_VAR
                  Reset := SUPER^.Reset();

Done               := FALSE;
Busy               := FALSE;
CommandBuffered    := FALSE;
CommandAborted     := FALSE;
CommandInterrupted := FALSE; 

                
END_METHOD
END_FUNCTION_BLOCK

/// Reads and writes specific configuration parameters on RC that are required for the RI to work
FUNCTION_BLOCK MC_ExchangeConfigurationFB EXTENDS RobotLibraryBaseEnableFB
// ------------------------------------------------------------------------- 
//  SRCI Robot Library                                                
// ------------------------------------------------------------------------- 
//                                                                           
//  Object:      ExchangeConfigurationFB                                       
//  Author:      Thorsten Brach                                                
//  Date:        2024-06-01
//
//  Description:                                              
//   
//                                                                           
//  Copyright: 
//    (C) 2024 Thorsten Brach. All rights reserved                                                                                                                                            
//             Licensed under the MIT License.
//                                                                           
//  Disclaimer:                                                                           
//    This project is provided without any guarantee and can be used for   
//    private and commercial purposes. Any use is at the user’s 
//    own risk and responsibility.
//
// -------------------------------------------------------------------------
VAR_INPUT
  /// Command parameter 
  ParCmd            : ExchangeConfigurationParCmd;
END_VAR

VAR_OUTPUT
  /// Command is transferred and confirmed by the RC
  CommandBuffered   : BOOL;
  /// Receiving of input parameter values has been acknowledged by RC
  ParameterAccepted : BOOL;
  /// command results
  OutCmd            : ExchangeConfigurationOutCmd;
END_VAR

VAR
  /// internal copy of command parameter 
 _parCmd            : ExchangeConfigurationParCmd;
  /// command data to send
 _command           : ExchangeConfigurationSendData;
  /// response data received
 _response          : ExchangeConfigurationRecvData;
END_VAR

            SUPER^(AxesGroup := AxesGroup);
          

METHOD INTERNAL CheckAddParameter : BOOL
VAR_INPUT
  /// Payload pointer
  PayloadPtr : UDINT;
END_VAR
VAR
  /// Payload as byte array
  Payload    : ARRAY [1..SIZEOF(_command)] OF BYTE;
  /// Null Byte array 
  Null       : ARRAY [1..SIZEOF(_command)] OF BYTE;
  /// Data length to compare
  DataLen    : UDINT;
END_VAR
                  // Payload pointer must be decreased by one byte, because ADR(Payload) is already one byte !
PayloadPtr := LIMIT (0, PayloadPtr - 1, SIZEOF(Payload) -1);
// Convert command struct to payload array
SysDepMemCpy( pDest := ADR(Payload), pSrc := ADR(_command), DataLen := SIZEOF(_command));
// Calculate the data length to compare - at least one byte must be compared !
DataLen := LIMIT(1, SIZEOF(Payload) - PayloadPtr, SIZEOF(Payload)); 
// Compare Payload-Array with Null-Byte-Array
CheckAddParameter := SysDepMemCmp( pData1 := ADR(Payload) + PayloadPtr , pData2 := ADR(Null), DataLen := DataLen) <>  RobotLibraryConstants.OK ;
                
END_METHOD

METHOD PROTECTED CheckFunctionSupported : BOOL
VAR_IN_OUT
  /// Robot assignment of function
  AxesGroup : AxesGroup; 
END_VAR
                  CheckFunctionSupported := TRUE; // Function is mandatory 
RETURN;

CheckFunctionSupported := AxesGroup.State.RobotData.RCSupportedFunctions.ExchangeConfiguration;

IF ( NOT CheckFunctionSupported )
THEN
  // call base implementation for set error and create log entry
  SUPER^.CheckFunctionSupported(AxesGroup := AxesGroup);
END_IF
                
END_METHOD

METHOD PROTECTED CheckParameterChanged : BOOL
VAR_IN_OUT
  /// Robot assignment of function
  AxesGroup    : AxesGroup; 
END_VAR
                  // Check ParCmd Size is > 0, because MemCmp does not work correctly with size = 0
IF (SIZEOF(ParCmd) = 0) OR (_stepCmd = 0)
THEN 
  RETURN;
END_IF

// compare memory 
_parameterChanged := ( SysDepMemCmp(pData1 := ADR(ParCmd), pData2 := ADR(_parCmd), DataLen := SIZEOF(ParCmd)) <> RobotLibraryConstants.OK );

// check parameter valid ?
_parameterValid   := CheckParameterValid( AxesGroup := AxesGroup );

IF ((  _parameterChanged        )  AND 
    (  _parameterValid          )) OR
    (  _parameterUpdateInternal )  
THEN  
  // Create log entry for parameter changed event
  CreateLogMessagePara1 ( Timestamp   := AxesGroup.State.SystemTime,
                          MessageType := MessageType.CMD,
                          Severity    := Severity.DEBUG,
                          MessageCode := 0,
                          MessageText := 'NotifyParameterChanged Event {1}',
                          Para1       :=  '' );

  // reset internal flag for send parameter update
 _parameterUpdateInternal := FALSE;
  // update internal copy of parameters 
 _parCmd := ParCmd;
  // inc parameter sequence
 _command.ParSeq := _command.ParSeq + 1;
  // update command data  
  CommandData := CreateCommandPayload(AxesGroup := AxesGroup); // ( Access via reference to rCommandFB in ACR )
  // notify active command register 
  AxesGroup.Acyclic.ActiveCommandRegister.NotifyParameterChanged := _uniqueID;
  // Reset parameter accepted flag
  ParameterAccepted := FALSE;
END_IF
                
END_METHOD

METHOD PROTECTED CheckParameterValid : BOOL
VAR_IN_OUT
  /// Robot assignment of function
  AxesGroup : AxesGroup; 
END_VAR
                  CheckParameterValid := TRUE;

// Check ParCmd.LogLevel valid ? 
IF (( ParCmd.LogLevel <> Severity.DEACTIVATE  ) AND  
    ( ParCmd.LogLevel <> Severity.DEBUG       ) AND
    ( ParCmd.LogLevel <> Severity.INFO        ) AND
    ( ParCmd.LogLevel <> Severity.WARNING     ) AND
    ( ParCmd.LogLevel <> Severity.ERROR       ) AND
    ( ParCmd.LogLevel <> Severity.FATAL_ERROR ))    
THEN
  // Parameter not valid
  CheckParameterValid := FALSE;
  // Set error
  SetError( ErrorID := RobotLibraryErrorIdEnum.ERR_INVALID_PAR_CMD, Overwrite := TRUE );
  // Create log entry
  CreateLogMessagePara1 ( Timestamp   := AxesGroup.State.SystemTime,
                          MessageType := MessageType.CMD,
                          Severity    := Severity.ERROR,
                          MessageCode := ErrorID,
                          MessageText := 'Invalid Parameter ParCmd.LogLevel = {1}',
                          Para1       :=  LOG_LEVEL_TO_STRING(ParCmd.LogLevel));
  RETURN;                          
END_IF


// Check ParCmd.WaitAtBlendingZone
// -> no plausibility check for boolean


// Check ParCmd.AllowSecSeqWhileSubprogram
// -> no plausibility check for boolean


// Check ParCmd.DelayTime valid ? 
IF ( ParCmd.DelayTime < 0  )   
THEN
  // Parameter not valid
  CheckParameterValid := FALSE;
  // Set error
  SetError( ErrorID := RobotLibraryErrorIdEnum.ERR_INVALID_PAR_CMD, Overwrite := TRUE );
  // Create log entry
  CreateLogMessagePara1 ( Timestamp   := AxesGroup.State.SystemTime,
                          MessageType := MessageType.CMD,
                          Severity    := Severity.ERROR,
                          MessageCode := ErrorID,
                          MessageText := 'Invalid Parameter ParCmd.DelayTime = {1} ms',
                          Para1       :=  UINT_TO_STRING(ParCmd.DelayTime));
  RETURN;                          
END_IF


// Check ParCmd.WaitForNrOfCmd valid ? 
IF ( ParCmd.WaitForNrOfCmd < 0  )   
THEN
  // Parameter not valid
  CheckParameterValid := FALSE;
  // Set error
  SetError( ErrorID := RobotLibraryErrorIdEnum.ERR_INVALID_PAR_CMD , Overwrite :=  TRUE );
  // Create log entry
  CreateLogMessagePara1 ( Timestamp   := AxesGroup.State.SystemTime,
                          MessageType := MessageType.CMD,
                          Severity    := Severity.ERROR,
                          MessageCode := ErrorID,
                          MessageText := 'Invalid Parameter ParCmd.WaitForNrOfCmd = {1}',
                          Para1       :=  UINT_TO_STRING(ParCmd.WaitForNrOfCmd));
  RETURN;                          
END_IF


// Check ParCmd.LifeSignTimeOut valid ? 
IF ( ParCmd.LifeSignTimeOut < 10 )   
THEN
  // Parameter not valid
  CheckParameterValid := FALSE;
  // Set error
  SetError( ErrorID := RobotLibraryErrorIdEnum.ERR_INVALID_PAR_CMD, Overwrite := TRUE );
  // Create log entry
  CreateLogMessagePara1 ( Timestamp   := AxesGroup.State.SystemTime,
                          MessageType := MessageType.CMD,
                          Severity    := Severity.ERROR,
                          MessageCode := ErrorID,
                          MessageText := 'Invalid Parameter ParCmd.LifeSignTimeOut = {1} ms',
                          Para1       :=  UINT_TO_STRING(ParCmd.LifeSignTimeOut));
  RETURN;                          
END_IF


// Check ParCmd.SyncDelay valid ? 
IF ( ParCmd.SyncDelay < 0  )   
THEN
  // Parameter not valid
  CheckParameterValid := FALSE;
  // Set error
  SetError( ErrorID := RobotLibraryErrorIdEnum.ERR_INVALID_PAR_CMD, Overwrite := TRUE ); 
  // Create log entry
  CreateLogMessagePara1 ( Timestamp   := AxesGroup.State.SystemTime,
                          MessageType := MessageType.CMD,
                          Severity    := Severity.ERROR,
                          MessageCode := ErrorID,
                          MessageText := 'Invalid Parameter ParCmd.SyncDelay = {1}',
                          Para1       :=  UINT_TO_STRING(ParCmd.SyncDelay));
  RETURN;                          
END_IF


// Check ParCmd.SyncReaction valid ? 
IF (( ParCmd.SyncReaction <> SyncReaction.NO_REACTION                      ) AND  
    ( ParCmd.SyncReaction <> SyncReaction.NO_AUTOMATIC_DISABLE             ) AND
    ( ParCmd.SyncReaction <> SyncReaction.INTERRUPT_WHEN_SEQUENCE_IS_EMPTY ) AND
    ( ParCmd.SyncReaction <> SyncReaction.IMMEDIATE_INTERRUPT              ))
THEN
  // Parameter not valid
  CheckParameterValid := FALSE;
  // Set error
  SetError( ErrorID := RobotLibraryErrorIdEnum.ERR_INVALID_PAR_CMD, Overwrite := TRUE ); 
  // Create log entry
  CreateLogMessagePara1 ( Timestamp   := AxesGroup.State.SystemTime,
                          MessageType := MessageType.CMD,
                          Severity    := Severity.ERROR,
                          MessageCode := ErrorID,
                          MessageText := 'Invalid Parameter ParCmd.SyncReaction = {1}',
                          Para1       :=  SYNC_REACTION_TO_STRING(ParCmd.SyncReaction));
  RETURN;                          
END_IF


// Check ParCmd.DataInSync.ToolsInSync
// -> no plausibility check for boolean


// Check ParCmd.DataInSync.FramesInSync
// -> no plausibility check for boolean


// Check ParCmd.DataInSync.LoadsInSync
// -> no plausibility check for boolean


// Check ParCmd.DataInSync.WorkAreasInSync
// -> no plausibility check for boolean


// Check ParCmd.DataInSync.SoftwareLimitsInSync
// -> no plausibility check for boolean


// Check ParCmd.DataInSync.DefaultDynamicsInSync
// -> no plausibility check for boolean


// Check ParCmd.DataInSync.ReferenceDynamicsInSync
// -> no plausibility check for boolean


// Check ParCmd.DataEnableSync.EnableSyncTool
// -> no plausibility check for boolean


// Check ParCmd.DataEnableSync.EnableSyncFrame
// -> no plausibility check for boolean


// Check ParCmd.DataEnableSync.EnableSyncLoad
// -> no plausibility check for boolean


// Check ParCmd.DataEnableSync.EnableSyncWorkArea
// -> no plausibility check for boolean


// Check ParCmd.DataEnableSync.EnableSyncSWLimits
// -> no plausibility check for boolean


// Check ParCmd.DataEnableSync.EnableSyncDefaultDynamics
// -> no plausibility check for boolean


// Check ParCmd.DataEnableSync.EnableSyncReferenceDynamics
// -> no plausibility check for boolean

// Check ParCmd.DataEnableSync.AllowDynamicBlending
// -> no plausibility check for boolean

                
END_METHOD

METHOD INTERNAL CreateCommandPayload : RobotLibraryCommandDataFB
VAR_IN_OUT
  /// Robot assignment of function
  AxesGroup  : AxesGroup; 
END_VAR
VAR
  /// Parameter count
 _parameterCnt : DINT;
END_VAR

// Table 6-86: Sent CMD payload (PLC to RC) of "ExchangeConfiguration"
// --------------------------
// Header
// --------------------------
// Byte 00 : UINT  - Type HB     
// Byte 01 :       - Type LB    
// Byte 02 : USINT - Reserve | ExecutionMode
// Byte 03 : USINT - ParSeq  | Priority
// --------------------------
// Datablock
// --------------------------
// Byte 4   : USINT      - LogLevel
// Byte 5.0 : BOOL       - WaitAtBlendingZone
// Byte 5.1 : BOOL       - Enable
// Byte 5.2 : BOOL       - AllowSecSeqWhileSubprogram
// Byte 5.3 : BOOL       - AllowDynamicBlending
// Byte 6   : UINT       - DelayTime HB
// Byte 7   :            - DelayTime LB
// Byte 8   : UINT       - WaitForNrOfCmd HB
// Byte 9   :            - WaitForNrOfCmd LB
// Byte 10  : UINT       - LifeSignTimeOut HB
// Byte 11  :            - LifeSignTimeOut LB
// Byte 12  : UINT       - SyncDelay HB
// Byte 13  :            - SyncDelay LB
// Byte 14  : USINT      - SyncReaction
// Byte 15  : BYTE       - Reserved
// Byte 16  : DataInSync - DataInSync 
// Byte 17  : BYTE       - Reserved
// Byte 18  : BYTE       - DataEnableSync
// Byte 19  : BYTE       - Reserved
                  // set command parameter 
_command.CmdTyp          :=  CmdType.ExchangeConfiguration;
_command.ExecMode        :=  ExecMode;
_command.ParSeq          := _command.ParSeq;
_command.Priority        :=  Priority;
_command.LogLevel        := _parCmd.LogLevel;
_command.CtrlByte.0      := _parCmd.WaitAtBlendingZone;
_command.CtrlByte.1      :=  Enable;
_command.CtrlByte.2      := _parCmd.AllowSecSeqWhileSubprogram;
_command.CtrlByte.3      := _parCmd.AllowDynamicBlending;
_command.DelayTime       := _parCmd.DelayTime;
_command.WaitForNrOfCmd  := _parCmd.WaitForNrOfCmd;
_command.LifeSignTimeOut := _parCmd.LifeSignTimeOut;
_command.SyncDelay       := _parCmd.SyncDelay;
_command.SyncReaction    := _parCmd.SyncReaction;
_command.Reserve1        := 0;
_command.DataInSync      := _parCmd.DataInSync;
_command.Reserve2        := 0;
_command.DataEnableSync  := _parCmd.DataEnableSync;  
_command.Reserve3        := 0;

// copy command data to header
_cmdHeader := _command;
// call base implementation to copy header to payload buffer
CreateCommandPayload := SUPER^.CreateCommandPayload(AxesGroup := AxesGroup);


// Check parameter must be added ? 
IF ( CheckAddParameter(CreateCommandPayload.PayloadPtr))
THEN
  // add command.LogLeve
  CreateCommandPayload.AddUsint(SINT_TO_USINT(_command.LogLevel));
  // inc parameter counter
 _parameterCnt := _parameterCnt + 1;  
END_IF


// Check parameter must be added ? 
IF ( CheckAddParameter(CreateCommandPayload.PayloadPtr))
THEN
  // add command.CtrlByte
  CreateCommandPayload.AddByte(_command.CtrlByte);
  // inc parameter counter
 _parameterCnt := _parameterCnt + 1;  
END_IF


// Check parameter must be added ? 
IF ( CheckAddParameter(CreateCommandPayload.PayloadPtr))
THEN
  // add command.DelayTime
  CreateCommandPayload.AddUint(_command.DelayTime);
  // inc parameter counter
 _parameterCnt := _parameterCnt + 1;  
END_IF


// Check parameter must be added ? 
IF ( CheckAddParameter(CreateCommandPayload.PayloadPtr))
THEN
  // add command.WaitForNrOfCmd
  CreateCommandPayload.AddUint(_command.WaitForNrOfCmd);
  // inc parameter counter
 _parameterCnt := _parameterCnt + 1;  
END_IF


// Check parameter must be added ? 
IF ( CheckAddParameter(CreateCommandPayload.PayloadPtr))
THEN
  // add command.LifeSignTimeOut
  CreateCommandPayload.AddUint(_command.LifeSignTimeOut);
  // inc parameter counter
 _parameterCnt := _parameterCnt + 1;  
END_IF


// Check parameter must be added ? 
IF ( CheckAddParameter(CreateCommandPayload.PayloadPtr))
THEN
  // add command.SyncDelay
  CreateCommandPayload.AddUint(_command.SyncDelay);
  // inc parameter counter
 _parameterCnt := _parameterCnt + 1;  
END_IF


// Check parameter must be added ? 
IF ( CheckAddParameter(CreateCommandPayload.PayloadPtr))
THEN
  // add command.SyncReaction
  CreateCommandPayload.AddUsint(_command.SyncReaction);
  // inc parameter counter
 _parameterCnt := _parameterCnt + 1;  
END_IF


// Check parameter must be added ? 
IF ( CheckAddParameter(CreateCommandPayload.PayloadPtr))
THEN
  // add command.SyncReaction
  CreateCommandPayload.AddUsint(_command.Reserve1);
  // inc parameter counter
 _parameterCnt := _parameterCnt + 1;  
END_IF


// Check parameter must be added ? 
IF ( CheckAddParameter(CreateCommandPayload.PayloadPtr))
THEN
  // add command.DataInSync
  CreateCommandPayload.AddDataInSync(_command.DataInSync);
  // inc parameter counter
 _parameterCnt := _parameterCnt + 1;  
END_IF


// Check parameter must be added ? 
IF ( CheckAddParameter(CreateCommandPayload.PayloadPtr))
THEN
  // add command.Reserve1
  CreateCommandPayload.AddByte(_command.Reserve2);
  // inc parameter counter
 _parameterCnt := _parameterCnt + 1;  
END_IF


// Check parameter must be added ? 
IF ( CheckAddParameter(CreateCommandPayload.PayloadPtr))
THEN
  // add command.DataEnableSync
  CreateCommandPayload.AddDataEnableSync(_command.DataEnableSync);
  // inc parameter counter
 _parameterCnt := _parameterCnt + 1;  
END_IF


// Check parameter must be added ? 
IF ( CheckAddParameter(CreateCommandPayload.PayloadPtr))
THEN
  // add command.Reserve2
  CreateCommandPayload.AddByte(_command.Reserve3);
  // inc parameter counter
 _parameterCnt := _parameterCnt + 1;  
END_IF


// Create logging
CreateCommandPayloadLog(AxesGroup := AxesGroup, ParameterCnt := _parameterCnt);
                
END_METHOD

METHOD INTERNAL CreateCommandPayloadLog
VAR_IN_OUT
  /// Robot assignment of function
  AxesGroup : AxesGroup; 
END_VAR
VAR_INPUT
  /// Parameter count
  ParameterCnt : DINT;
END_VAR
                  // Create log entry for Parameter start
CreateLogMessagePara1 ( Timestamp   := AxesGroup.State.SystemTime,
                        MessageType := MessageType.CMD,
                        Severity    := Severity.DEBUG,
                        MessageCode := 0,
                        MessageText := 'Create command payload with {1} parameter(s) :',
                        Para1       := DINT_TO_STRING(ParameterCnt));
  

// Return if no parameter is remaining...
IF ( ParameterCnt = 0 ) THEN RETURN; END_IF
// dec remaining parameter(s)                        
ParameterCnt := ParameterCnt - 1;
// Create log entry for LogLevel
CreateLogMessagePara1 ( Timestamp   := AxesGroup.State.SystemTime,
                        MessageType := MessageType.CMD,
                        Severity    := Severity.DEBUG,
                        MessageCode := 0,
                        MessageText := 'Command.LogLevel = {1}',
                        Para1       :=  LOG_LEVEL_TO_STRING(_command.LogLevel));


// Return if no parameter is remaining...
IF ( ParameterCnt = 0 ) THEN RETURN; END_IF
// dec remaining parameter(s)                        
ParameterCnt := ParameterCnt - 1;
// Create log entry for CtrlByte
CreateLogMessagePara1 ( Timestamp   := AxesGroup.State.SystemTime,
                        MessageType := MessageType.CMD,
                        Severity    := Severity.DEBUG,
                        MessageCode := 0,
                        MessageText := 'Command.CtrlByte = {1}',
                        Para1       :=  BYTE_TO_STRING(_command.CtrlByte));


// Return if no parameter is remaining...
IF ( ParameterCnt = 0 ) THEN RETURN; END_IF
// dec remaining parameter(s)                        
ParameterCnt := ParameterCnt - 1;
// Create log entry for DelayTime
CreateLogMessagePara1 ( Timestamp   := AxesGroup.State.SystemTime,
                        MessageType := MessageType.CMD,
                        Severity    := Severity.DEBUG,
                        MessageCode := 0,
                        MessageText := 'Command.DelayTime = {1}',
                        Para1       :=  UINT_TO_STRING(_command.DelayTime));


// Return if no parameter is remaining...
IF ( ParameterCnt = 0 ) THEN RETURN; END_IF
// dec remaining parameter(s)                        
ParameterCnt := ParameterCnt - 1;
// Create log entry for WaitForNrOfCmd
CreateLogMessagePara1 ( Timestamp   := AxesGroup.State.SystemTime,
                        MessageType := MessageType.CMD,
                        Severity    := Severity.DEBUG,
                        MessageCode := 0,
                        MessageText := 'Command.WaitForNrOfCmd = {1}',
                        Para1       :=  UINT_TO_STRING(_command.WaitForNrOfCmd));


// Return if no parameter is remaining...
IF ( ParameterCnt = 0 ) THEN RETURN; END_IF
// dec remaining parameter(s)                        
ParameterCnt := ParameterCnt - 1;
// Create log entry for LifeSignTimeOut
CreateLogMessagePara1 ( Timestamp   := AxesGroup.State.SystemTime,
                        MessageType := MessageType.CMD,
                        Severity    := Severity.DEBUG,
                        MessageCode := 0,
                        MessageText := 'Command.LifeSignTimeOut = {1}',
                        Para1       :=  UINT_TO_STRING(_command.LifeSignTimeOut));


// Return if no parameter is remaining...
IF ( ParameterCnt = 0 ) THEN RETURN; END_IF
// dec remaining parameter(s)                        
ParameterCnt := ParameterCnt - 1;
// Create log entry for SyncDelay
CreateLogMessagePara1 ( Timestamp   := AxesGroup.State.SystemTime,
                        MessageType := MessageType.CMD,
                        Severity    := Severity.DEBUG,
                        MessageCode := 0,
                        MessageText := 'Command.SyncDelay = {1}',
                        Para1       :=  UINT_TO_STRING(_command.SyncDelay));


// Return if no parameter is remaining...
IF ( ParameterCnt = 0 ) THEN RETURN; END_IF
// dec remaining parameter(s)                        
ParameterCnt := ParameterCnt - 1;
// Create log entry for SyncReaction
CreateLogMessagePara1 ( Timestamp   := AxesGroup.State.SystemTime,
                        MessageType := MessageType.CMD,
                        Severity    := Severity.DEBUG,
                        MessageCode := 0,
                        MessageText := 'Command.SyncReaction = {1}',
                        Para1       :=  SYNC_REACTION_TO_STRING(_command.SyncReaction));


// Return if no parameter is remaining...
IF ( ParameterCnt = 0 ) THEN RETURN; END_IF
// dec remaining parameter(s)                        
ParameterCnt := ParameterCnt - 1;
// Create log entry for Reserve1
CreateLogMessagePara1 ( Timestamp   := AxesGroup.State.SystemTime,
                        MessageType := MessageType.CMD,
                        Severity    := Severity.DEBUG,
                        MessageCode := 0,
                        MessageText := 'Command.Reserve1 = {1}',
                        Para1       :=  BYTE_TO_STRING(_command.Reserve1));



// Return if no parameter is remaining...
IF ( ParameterCnt = 0 ) THEN RETURN; END_IF
// dec remaining parameter(s)                        
ParameterCnt := ParameterCnt - 1;
// Create log entry for DataInSync
CreateLogMessagePara1 ( Timestamp   := AxesGroup.State.SystemTime,
                        MessageType := MessageType.CMD,
                        Severity    := Severity.DEBUG,
                        MessageCode := 0,
                        MessageText := 'Command.DataInSync = {1}',
                        Para1       :=  DATA_IN_SYNC_TO_STRING(_command.DataInSync));


// Return if no parameter is remaining...
IF ( ParameterCnt = 0 ) THEN RETURN; END_IF
// dec remaining parameter(s)                        
ParameterCnt := ParameterCnt - 1;
// Create log entry for Reserve1
CreateLogMessagePara1 ( Timestamp   := AxesGroup.State.SystemTime,
                        MessageType := MessageType.CMD,
                        Severity    := Severity.DEBUG,
                        MessageCode := 0,
                        MessageText := 'Command.Reserve2 = {1}',
                        Para1       :=  BYTE_TO_STRING(_command.Reserve2));


// Return if no parameter is remaining...
IF ( ParameterCnt = 0 ) THEN RETURN; END_IF
// dec remaining parameter(s)                        
ParameterCnt := ParameterCnt - 1;
// Create log entry for DataEnableSync
CreateLogMessagePara1 ( Timestamp   := AxesGroup.State.SystemTime,
                        MessageType := MessageType.CMD,
                        Severity    := Severity.DEBUG,
                        MessageCode := 0,
                        MessageText := 'Command.DataEnableSync = {1}',
                        Para1       :=  DATA_ENABLE_SYNC_TO_STRING(_command.DataEnableSync));


// Return if no parameter is remaining...
IF ( ParameterCnt = 0 ) THEN RETURN; END_IF
// dec remaining parameter(s)                        
ParameterCnt := ParameterCnt - 1;
// Create log entry for Reserve2
CreateLogMessagePara1 ( Timestamp   := AxesGroup.State.SystemTime,
                        MessageType := MessageType.CMD,
                        Severity    := Severity.DEBUG,
                        MessageCode := 0,
                        MessageText := 'Command.Reserve3 = {1}',
                        Para1       :=  BYTE_TO_STRING(_command.Reserve3));
                
END_METHOD

METHOD FB_init : BOOL
VAR_INPUT
  /// if TRUE, the retain variables are initialized (warm start / cold start)
  bInitRetains : BOOL; 
  /// if TRUE, the instance afterwards gets moved into the copy code (online change)
  bInCopyCode  : BOOL;  
END_VAR
                  MyType   := 'MC_ExchangeConfigurationFB';
ExecMode := ExecutionMode.PARALLEL;
Priority := PriorityLevel.NORMAL;
                
END_METHOD

METHOD PROTECTED OnApplyOutCmd
VAR_INPUT
  /// Command message state
  State : CmdMessageState;
END_VAR
                  IF ( State = CmdMessageState.EMPTY ) 
THEN
  // Reset command outputs
  SysDepMemSet(pDest := ADR(OutCmd), Value := 0, DataLen := SIZEOF(OutCmd));         
END_IF

IF ( State = CmdMessageState.ACTIVE ) OR ( TRUE )
THEN  
  // Update command outputs
  OutCmd.LengthACR                 := _response.LengthACR;
  OutCmd.HighestToolIndex          := _response.HighestToolIndex;
  OutCmd.HighestFrameIndex         := _response.HighestFrameIndex;
  OutCmd.HighestLoadIndex          := _response.HighestLoadIndex;
  OutCmd.HighestWorkAreaIndex      := _response.HighestWorkAreaIndex;
  OutCmd.DataInSync                := _response.DataInSync;
  OutCmd.ChangeIndexTool           := _response.ChangeIndexTool;
  OutCmd.ChangeIndexFrame          := _response.ChangeIndexFrame;
  OutCmd.ChangeIndexLoad           := _response.ChangeIndexLoad;
  OutCmd.ChangeIndexWorkArea       := _response.ChangeIndexWorkArea;
  OutCmd.RAWorkingHours            := _response.RAWorkingHours;
  OutCmd.BrakeTestRequired         := _response.StatusByte.0;
  OutCmd.StepModeExactStopActive   := _response.StatusByte.1;
  OutCmd.StepModeBlendingActive    := _response.StatusByte.2;
  OutCmd.PathAccuracyMode          := _response.StatusByte.3;
  OutCmd.AvoidSingularity          := _response.StatusByte.4;
  OutCmd.CollisionDetectionEnabled := _response.StatusByte.5;
  OutCmd.AcceleratingSupported     := _response.StatusByte.6;
  OutCmd.DecceleratingSupported    := _response.StatusByte.7;
  OutCmd.ConstantVelocitySupported := _response.ConstantVelocitySupported;
  OutCmd.RCWorkingHours            := _response.RCWorkingHours;      
END_IF
                
END_METHOD

METHOD Protected OnExecCancel : DINT
VAR_IN_OUT
  /// Robot assignment of function
  AxesGroup : AxesGroup; 
END_VAR
VAR
  /// internal return value 
 _retVal    : DINT;
END_VAR
                  OnExecCancel := RobotLibraryConstants.RUNNING;

CASE _stepCancel OF
  
  0: // set busy flag
     Busy := TRUE;
    
     // Create log entry
     CreateLogMessagePara1 ( Timestamp   := AxesGroup.State.SystemTime,
                             MessageType := MessageType.CMD,
                             Severity    := Severity.DEBUG,
                             MessageCode := 0,
                             MessageText := 'Execution of {1} cancelled',
                             Para1       := MyType);                 
    
     // try to remove cmd
    _retVal := AxesGroup.Acyclic.ActiveCommandRegister.RemoveCmd(_uniqueID);
  
     // check result of removement       
     IF ( _retVal = RobotLibraryConstants.OK )
     THEN
       // Reset step counter
      _stepCancel := 0;
       // finished okay
       OnExecCancel := RobotLibraryConstants.OK;
     
       // Create log entry
       CreateLogMessagePara1 ( Timestamp   := AxesGroup.State.SystemTime,
                               MessageType := MessageType.CMD,
                               Severity    := Severity.DEBUG,
                               MessageCode := 0,
                               MessageText := '{1} successfully removed from ACR',
                               Para1       := MyType);                 
     ELSE
       // set timeout
       SetTimeout(PT := _timeoutCancel, rTimer := _timerCancel);
       // inc step counter
      _stepCancel := _stepCancel + 1; 
     
       // Create log entry
       CreateLogMessagePara1 ( Timestamp   := AxesGroup.State.SystemTime,
                               MessageType := MessageType.CMD,
                               Severity    := Severity.DEBUG,
                               MessageCode := 0,
                               MessageText := '{1} was not removed from ACR because execution was already in progress',
                               Para1       := MyType);                 
     END_IF       
  
     
 1:  // call clear error 
     OnExecCancel := OnExecErrorClear(AxesGroup := AxesGroup);  
 
     IF ( OnExecCancel = RobotLibraryConstants.OK)
     THEN
       // Reset busy flag
       Busy := FALSE;
       // Reset step counter
      _stepCancel := 0;
       // finished okay
       OnExecCancel := RobotLibraryConstants.OK;
     END_IF  
  
ELSE
  // invalid step
  SetError( ErrorID := RobotLibraryErrorIdEnum.ERR_INVALID_STEP, Overwrite := TRUE );
END_CASE  


                        
// reset step counter
IF (OnExecCancel <> RobotLibraryConstants.RUNNING)
THEN
  // Reset FB variables
  Reset();
  // Reset step counter
 _stepCancel := 0;
END_IF                        
                
END_METHOD

METHOD PROTECTED OnExecErrorClear : DINT
VAR_IN_OUT
  /// Robot assignment of function
  AxesGroup : AxesGroup; 
END_VAR
                  OnExecErrorClear := RobotLibraryConstants.RUNNING;

CASE _stepClearError OF
  
  0:  // set busy flag
      Busy := TRUE;
      // trigger parameter update to disable FB
     _parameterUpdateInternal := TRUE;
      // call Check Parameter changed method to trigger the parameter update to disable the function
      CheckParameterChanged(AxesGroup := AxesGroup);
      // set timeout
      SetTimeout(PT := _timeoutClearError, rTimer := _timerClearError);
      // inc step counter
     _stepClearError := _stepClearError + 1; 
      
  1: IF ( _responseReceived )
     THEN
       // reset response received flag
      _responseReceived := FALSE;
       // reset step counter
      _stepClearError := 0;
       // finished
       OnExecErrorClear := RobotLibraryConstants.OK;
     ELSE
       // timeout exceeded ? 
       IF (CheckTimeout(_timerClearError) = RobotLibraryConstants.OK)
       THEN
         OnExecErrorClear := RobotLibraryConstants.HAS_ERROR;
       END_IF
	   END_IF
ELSE
  // invalid step
  SetError( ErrorID := RobotLibraryErrorIdEnum.ERR_INVALID_STEP, Overwrite := TRUE );
END_CASE


// reset step counter
IF (OnExecErrorClear <> RobotLibraryConstants.RUNNING)
THEN
  // Reset 
  Reset();     
  // reset step counter
 _stepClearError := 0;
END_IF
                
END_METHOD

METHOD PROTECTED OnExecRun : DINT
VAR_IN_OUT
  /// Robot assignment of function
  AxesGroup : AxesGroup; 
END_VAR
                  // call base implementation
SUPER^.OnExecRun(AxesGroup := AxesGroup);


CASE _stepCmd OF
  
  00:  IF ( _enable_R.Q ) AND ( NOT Error) 
       THEN
         // reset the rising edge
        _enable_R();       

         // Check function is supported and parameter are valid ?
         IF (( CheckFunctionSupported( AxesGroup := AxesGroup )) AND
             ( CheckParameterValid   ( AxesGroup := AxesGroup )))      
         THEN
           // Reset all internal flags
           Reset();
           // set busy flag
           Busy := TRUE;
           // Reset command outputs
           SysDepMemSet(pDest := ADR(OutCmd), Value := 0, DataLen := SIZEOF(OutCmd));         
           // apply command parameter
          _parCmd := ParCmd;
           // init parameter sequence
          _command.ParSeq := 1;
           // create command data
           CommandData := CreateCommandPayload(AxesGroup := AxesGroup);
           // Add command to active command register
          _uniqueID := AxesGroup.Acyclic.ActiveCommandRegister.AddCmd( pCommandFB := ADR(THIS^ ));     
           // set timeout
           SetTimeout(PT := _timeoutCmd, rTimer := _timerCmd);
           // inc step counter
          _stepCmd := _stepCmd + 1; 
         END_IF
       END_IF
     

  01:  // Wait for responce received
       IF ( _responseReceived )
       THEN
         // reset response received flag
        _responseReceived := FALSE;
         // update state flags
         OnUpdateStateFlags(_response.State);
         // update state flags
         OnApplyOutCmd(_response.State);
       END_IF

       // do not abort directly, so that the ParSeq update can be send
       IF ( _enable_F.Q ) 
       THEN
         // Reset Enabled Flag
         Enabled := FALSE;
         // Set Busy flag
         Busy := TRUE;
         // trigger parameter update to disable FB
        _parameterUpdateInternal := TRUE;
         // reset the falling edge
        _enable_F();
         // set timeout
         SetTimeout(PT := _timeoutCmd, rTimer := _timerCmd);
         // inc step counter
        _stepCmd := _stepCmd + 1; 
       END_IF

  02: IF ((    _responseReceived                                   )  OR 
          (     CheckTimeout(_timerCmd) = RobotLibraryConstants.OK )) OR 
         (( NOT AxesGroup.State.Initialized                        )  AND
          ( NOT AxesGroup.State.Synchronized                       ))
      THEN
        Reset();   
	    END_IF
      
ELSE
  // invalid step
  SetError( ErrorID := RobotLibraryErrorIdEnum.ERR_INVALID_STEP, Overwrite := TRUE );
END_CASE



// Reset FB
IF (( _enable_R.Q ) OR
    ( _enable_F.Q ))
THEN
  Reset();
END_IF
                
END_METHOD

METHOD PROTECTED OnUpdateStateFlags
VAR_INPUT
  /// Command message state
  State : CmdMessageState;
END_VAR
                  // Reset State flags
;

// Update Enabled flag
Enabled := _response.Enabled OR State = CmdMessageState.ACTIVE; {warning 'ToDo: Stäubli send Enabled = FALSE instead of true'}

CASE State OF

  // No operation or process is active
  CmdMessageState.EMPTY               :;
  // Created but not yet started
  CmdMessageState.CREATED             :;
  // Buffered and awaiting execution
  CmdMessageState.BUFFERED            : CommandBuffered    := TRUE;
                                        ParameterAccepted  := TRUE;
  // Buffered in planner for future execution
  CmdMessageState.BUFFERED_IN_PLANNER : CommandBuffered    := TRUE;
                                        ParameterAccepted  := TRUE;
  // Currently active and in progress
  CmdMessageState.ACTIVE              : 
  // Interrupted and awaiting continuation
  CmdMessageState.INTERRUPTED         :;
  // Requested for abort
  CmdMessageState.ABORT_REQUEST       :;
  // Successfully completed
  CmdMessageState.DONE                : Busy  := FALSE;
  // Aborted before completion
  CmdMessageState.ABORTED             : Busy  := FALSE;
  // Encountered an error during execution
  CmdMessageState.ERROR               : Error := TRUE;
                                        Busy  := FALSE;
END_CASE
                
END_METHOD

METHOD INTERNAL ParseResponsePayload : DINT
VAR_INPUT
  /// Response data
  ResponseData : RobotLibraryResponseDataFB;
  /// Timestamp
  Timestamp    : SystemTime;  
END_VAR
VAR
  /// Parameter count
 _parameterCnt : DINT;
END_VAR

// Table 6-87: Received CMD payload (RC to PLC) of "ExchangeConfiguration"
// --------------------------
// Header
// --------------------------
// Byte 00 : USINT - ParSeq | State     
// Byte 01 : SINT  - AlarmMessageSeverity    
// Byte 02 : UINT  - AlarmMessageCode HB
// Byte 03 :       - AlarmMessageCode LB
// --------------------------
// Datablock
// --------------------------
// Byte 04 : BOOL       - Enabled
// Byte 05 : BYTE       - Reserve
// Byte 05 : UINT       - LengthACR LW HB
// Byte 06 :            - LengthACR LW LB
// Byte 08 : USINT      - HighestToolIndex
// Byte 09 : USINT      - HighestFrameIndex
// Byte 10 : USINT      - HighestLoadIndex
// Byte 11 : USINT      - HighestWorkAreaIndex
// Byte 12 : DataInSync - DataInSync
// Byte 13 : BYTE       - Reserve
// Byte 14 : USINT      - ChangeIndexTool
// Byte 15 : USINT      - ChangeIndexFrame
// Byte 16 : USINT      - ChangeIndexLoad
// Byte 17 : USINT      - ChangeIndexWorkArea
// Byte 18 : UDINT      - RA WorkingHours HW HB
// Byte 19 :            - RA WorkingHours HW LB
// Byte 20 :            - RA WorkingHours LW HB
// Byte 21 :            - RA WorkingHours LW LB
// Byte 22 : BYTE       - StatusByte
// Byte 23 : BOOL       - ConstantVelocitySupported
// Byte 24 : UDINT      - RC WorkingHours HW HB
// Byte 25 :            - RC WorkingHours HW LB
// Byte 26 :            - RC WorkingHours LW HB
// Byte 27 :            - RC WorkingHours LW LB
// --------------------------
                  // call base implementation to parse the header from payload buffer
ResponseData.PayloadPtr := SUPER^.ParseResponsePayload(ResponseData := ResponseData, Timestamp := Timestamp);

// copy parsed header to response
_response.ParSeq               := _rspHeader.ParSeq;
_response.State                := _rspHeader.State;
_response.AlarmMessageSeverity := _rspHeader.AlarmMessageSeverity;
_response.AlarmMessageCode     := _rspHeader.AlarmMessageCode;


// Check payload remaining ? 
IF ( ResponseData.IsPayloadRemaining)
THEN
  // Get Response.Enabled
 _response.Enabled := ResponseData.GetBool();
  // inc parameter counter
 _parameterCnt := _parameterCnt + 1;
END_IF


// Check payload remaining ? 
IF ( ResponseData.IsPayloadRemaining)
THEN
  // Get Response.Reserve1
 _response.Reserve1 := ResponseData.GetByte();
  // inc parameter counter
 _parameterCnt := _parameterCnt + 1;
END_IF


// Check payload remaining ? 
IF ( ResponseData.IsPayloadRemaining)
THEN
  // Get Response.LengthACR
 _response.LengthACR := ResponseData.GetUint();
  // inc parameter counter
 _parameterCnt := _parameterCnt + 1;
END_IF


// Check payload remaining ? 
IF ( ResponseData.IsPayloadRemaining)
THEN
  // Get Response.HighestToolIndex
 _response.HighestToolIndex := ResponseData.GetUsint();
  // inc parameter counter
 _parameterCnt := _parameterCnt + 1;
END_IF


// Check payload remaining ? 
IF ( ResponseData.IsPayloadRemaining)
THEN
  // Get Response.HighestFrameIndex
 _response.HighestFrameIndex := ResponseData.GetUsint();
  // inc parameter counter
 _parameterCnt := _parameterCnt + 1;
END_IF


// Check payload remaining ? 
IF ( ResponseData.IsPayloadRemaining)
THEN
  // Get Response.HighestLoadIndex
 _response.HighestLoadIndex := ResponseData.GetUsint();
  // inc parameter counter
 _parameterCnt := _parameterCnt + 1;
END_IF


// Check payload remaining ? 
IF ( ResponseData.IsPayloadRemaining)
THEN
  // Get Response.HighestWorkAreaIndex
 _response.HighestWorkAreaIndex := ResponseData.GetUsint();
  // inc parameter counter
 _parameterCnt := _parameterCnt + 1;
END_IF 


// Check payload remaining ? 
IF ( ResponseData.IsPayloadRemaining)
THEN
  // Get Response.DataInSync
 _response.DataInSync := ResponseData.GetDataInSync();
  // inc parameter counter
 _parameterCnt := _parameterCnt + 1;
END_IF 


// Check payload remaining ? 
IF ( ResponseData.IsPayloadRemaining)
THEN
  // Get Response.Reserve2
 _response.Reserve2 := ResponseData.GetByte();
  // inc parameter counter
 _parameterCnt := _parameterCnt + 1;
END_IF 


// Check payload remaining ? 
IF ( ResponseData.IsPayloadRemaining)
THEN
  // Get Response.ChangeIndexTool
 _response.ChangeIndexTool := ResponseData.GetUsint();
  // inc parameter counter
 _parameterCnt := _parameterCnt + 1;
END_IF 


// Check payload remaining ? 
IF ( ResponseData.IsPayloadRemaining)
THEN
  // Get Response.ChangeIndexFrame
 _response.ChangeIndexFrame := ResponseData.GetUsint();
  // inc parameter counter
 _parameterCnt := _parameterCnt + 1;
END_IF 


// Check payload remaining ? 
IF ( ResponseData.IsPayloadRemaining)
THEN
  // Get Response.ChangeIndexLoad
 _response.ChangeIndexLoad := ResponseData.GetUsint();
  // inc parameter counter
 _parameterCnt := _parameterCnt + 1;
END_IF 


// Check payload remaining ? 
IF ( ResponseData.IsPayloadRemaining)
THEN
  // Get Response.ChangeIndexWorkArea
 _response.ChangeIndexWorkArea := ResponseData.GetUsint();
  // inc parameter counter
 _parameterCnt := _parameterCnt + 1;
END_IF 


// Check payload remaining ? 
IF ( ResponseData.IsPayloadRemaining)
THEN
  // Get Response.RAWorkingHours
 _response.RAWorkingHours := ResponseData.GetUdint();
  // inc parameter counter
 _parameterCnt := _parameterCnt + 1;
END_IF 


// Check payload remaining ? 
IF ( ResponseData.IsPayloadRemaining)
THEN
  // Get Response.StatusByte
 _response.StatusByte := ResponseData.GetByte();
  // inc parameter counter
 _parameterCnt := _parameterCnt + 1;
END_IF 


// Check payload remaining ? 
IF ( ResponseData.IsPayloadRemaining)
THEN
  // Get Response.ConstantVelocitySupported
 _response.ConstantVelocitySupported := ResponseData.GetBool();
  // inc parameter counter
 _parameterCnt := _parameterCnt + 1;
END_IF 


// Check payload remaining ? 
IF ( ResponseData.IsPayloadRemaining)
THEN
  // Get Response.RCWorkingHours
 _response.RCWorkingHours := ResponseData.GetUdint();
  // inc parameter counter
 _parameterCnt := _parameterCnt + 1;
END_IF 

// Create logging
ParseResponsePayloadLog(ResponseData := ResponseData, Timestamp := Timestamp, ParameterCnt := _parameterCnt);
                
END_METHOD

METHOD INTERNAL ParseResponsePayloadLog
VAR_INPUT
  /// Response data
  ResponseData : RobotLibraryResponseDataFB;
  /// Timestamp
  Timestamp    : SystemTime;  
  /// Parameter count
  ParameterCnt : DINT;
END_VAR
                  // Create log entry for Parameter start
CreateLogMessagePara1 ( Timestamp   := Timestamp,
                        MessageType := MessageType.CMD,
                        Severity    := Severity.DEBUG,
                        MessageCode := 0,
                        MessageText := '{1} parameter(s) to parse from the response data:',
                        Para1       := DINT_TO_STRING(ParameterCnt));


// Return if no parameter is remaining...
IF ( ParameterCnt = 0 ) THEN RETURN; END_IF
// dec remaining parameter(s)                        
ParameterCnt := ParameterCnt - 1;
// Create log entry for Enabled
CreateLogMessagePara1 ( Timestamp   := Timestamp,
                        MessageType := MessageType.CMD,
                        Severity    := Severity.DEBUG,
                        MessageCode := 0,
                        MessageText := 'Response.Enabled = {1}',
                        Para1       :=  BOOL_TO_STRING(_response.Enabled));


// Return if no parameter is remaining...
IF ( ParameterCnt = 0 ) THEN RETURN; END_IF
// dec remaining parameter(s)                        
ParameterCnt := ParameterCnt - 1;
// Create log entry for Reserve1
CreateLogMessagePara1 ( Timestamp   := Timestamp,
                        MessageType := MessageType.CMD,
                        Severity    := Severity.DEBUG,
                        MessageCode := 0,
                        MessageText := 'Response.Reserve1 = {1}',
                        Para1       :=  BYTE_TO_STRING(_response.Reserve1));


